LIN {X 0,Y 370.403,Z 508.31,A -85,B 0,C 180,E1 -12846.518,E2 -12846.518} C_VEL
LIN {X 0,Y 369.46,Z 515.734,A -85,B 0,C 180,E1 -12848.226,E2 -12848.226} C_VEL
LIN {X 0,Y 368.707,Z 521.584,A -85,B 0,C 180,E1 -12849.933,E2 -12849.933} C_VEL
LIN {X 0,Y 368.18,Z 526.14,A -85,B 0,C 180,E1 -12851.641,E2 -12851.641} C_VEL
LIN {X 0,Y 367.773,Z 529.554,A -85,B 0,C 180,E1 -12853.342,E2 -12853.342} C_VEL
LIN {X 0,Y 367.548,Z 531.232,A -85,B 0,C 180,E1 -12854.472,E2 -12854.472} C_VEL
LIN {X 0,Y 367.413,Z 532.492,A -85,B 0,C 180,E1 -12855.601,E2 -12855.601} C_VEL
LIN {X 0,Y 367.378,Z 533.578,A -85,B 0,C 180,E1 -12857.329,E2 -12857.329} C_VEL
LIN {X 0,Y 367.326,Z 533.705,A -85,B 0,C 180,E1 -12858.969,E2 -12858.969} C_VEL
LIN {X 0,Y 367.25,Z 533.313,A -85,B 0,C 180,E1 -12860.082,E2 -12860.082} C_VEL
LIN {X 0,Y 367.304,Z 532.493,A -85,B 0,C 180,E1 -12861.194,E2 -12861.194} C_VEL
LIN {X 0,Y 367.39,Z 531.247,A -85,B 0,C 180,E1 -12862.304,E2 -12862.304} C_VEL
LIN {X 0,Y 367.565,Z 528.8,A -85,B 0,C 180,E1 -12863.864,E2 -12863.864} C_VEL
LIN {X 0,Y 367.773,Z 524.966,A -85,B 0,C 180,E1 -12865.615,E2 -12865.615} C_VEL
LIN {X 0,Y 368.12,Z 520.21,A -85,B 0,C 180,E1 -12867.264,E2 -12867.264} C_VEL
LIN {X 0,Y 368.489,Z 514.221,A -85,B 0,C 180,E1 -12868.906,E2 -12868.906} C_VEL
LIN {X 0,Y 369.298,Z 506.742,A -85,B 0,C 180,E1 -12870.544,E2 -12870.544} C_VEL
LIN {X 0,Y 369.887,Z 499.149,A -85,B 0,C 180,E1 -12871.905,E2 -12871.905} C_VEL
LIN {X 0,Y 370.631,Z 489.936,A -85,B 0,C 180,E1 -12873.26,E2 -12873.26} C_VEL
LIN {X 0,Y 371.696,Z 479.626,A -85,B 0,C 180,E1 -12874.473,E2 -12874.473} C_VEL
LIN {X 0,Y 372.523,Z 468.25,A -85,B 0,C 180,E1 -12875.548,E2 -12875.548} C_VEL
LIN {X 0,Y 373.196,Z 456.407,A -85,B 0,C 180,E1 -12876.419,E2 -12876.419} C_VEL
LIN {X 0,Y 373.788,Z 443.261,A -85,B 0,C 180,E1 -12877.121,E2 -12877.121} C_VEL
LIN {X 0,Y 374.267,Z 430.141,A -85,B 0,C 180,E1 -12877.586,E2 -12877.586} C_VEL
LIN {X 0,Y 375.188,Z 377.579,A -85,B 0,C 180,E1 -12878.607,E2 -12878.607} C_VEL
LIN {X 0,Y 374.513,Z 369.843,A -85,B 0,C 180,E1 -12878.79,E2 -12878.79} C_VEL
LIN {X 0,Y 372.713,Z 362.305,A -85,B 0,C 180,E1 -12879.023,E2 -12879.023} C_VEL
LIN {X 0,Y 368.624,Z 347.244,A -85,B 0,C 180,E1 -12879.519,E2 -12879.519} C_VEL
LIN {X 0,Y 364.25,Z 322.715,A -85,B 0,C 180,E1 -12880.254,E2 -12880.254} C_VEL
LIN {X 0,Y 362.06,Z 310.498,A -85,B 0,C 180,E1 -12883.469,E2 -12883.469} C_VEL
LIN {X 0,Y 361.922,Z 310.404,A -85,B 0,C 180,E1 -12887.914,E2 -12887.914} C_VEL
LIN {X 0,Y 361.861,Z 310.408,A -85,B 0,C 180,E1 -12891.654,E2 -12891.654} C_VEL
LIN {X 0,Y 361.866,Z 310.405,A -85,B 0,C 180,E1 -12895.294,E2 -12895.294} C_VEL
LIN {X 0,Y 361.855,Z 310.407,A -85,B 0,C 180,E1 -12899.072,E2 -12899.072} C_VEL
LIN {X 0,Y 361.845,Z 310.41,A -85,B 0,C 180,E1 -12902.944,E2 -12902.944} C_VEL
LIN {X 0,Y 361.861,Z 310.406,A -85,B 0,C 180,E1 -12905.636,E2 -12905.636} C_VEL
LIN {X 0,Y 361.822,Z 310.414,A -85,B 0,C 180,E1 -12909.017,E2 -12909.017} C_VEL
LIN {X 0,Y 361.825,Z 310.418,A -85,B 0,C 180,E1 -12912.829,E2 -12912.829} C_VEL
LIN {X 0,Y 361.809,Z 310.412,A -85,B 0,C 180,E1 -12915.946,E2 -12915.946} C_VEL
LIN {X 0,Y 361.805,Z 310.417,A -85,B 0,C 180,E1 -12919.248,E2 -12919.248} C_VEL
LIN {X 0,Y 361.855,Z 310.411,A -85,B 0,C 180,E1 -12922.98,E2 -12922.98} C_VEL
LIN {X 0,Y 361.851,Z 310.408,A -85,B 0,C 180,E1 -12926.63,E2 -12926.63} C_VEL
LIN {X 0,Y 361.84,Z 310.412,A -85,B 0,C 180,E1 -12929.668,E2 -12929.668} C_VEL
LIN {X 0,Y 361.846,Z 310.415,A -85,B 0,C 180,E1 -12933.466,E2 -12933.466} C_VEL
LIN {X 0,Y 361.866,Z 310.407,A -85,B 0,C 180,E1 -12937.143,E2 -12937.143} C_VEL
LIN {X 0,Y 361.851,Z 310.407,A -85,B 0,C 180,E1 -12940.72,E2 -12940.72} C_VEL
LIN {X 0,Y 361.87,Z 310.407,A -85,B 0,C 180,E1 -12944.222,E2 -12944.222} C_VEL
LIN {X 0,Y 361.955,Z 310.395,A -85,B 0,C 180,E1 -12946.526,E2 -12946.526} C_VEL
LIN {X 0,Y 361.985,Z 310.397,A -85,B 0,C 180,E1 -12949.936,E2 -12949.936} C_VEL
LIN {X 0,Y 362.112,Z 310.375,A -85,B 0,C 180,E1 -12953.312,E2 -12953.312} C_VEL
LIN {X 0,Y 362.259,Z 310.358,A -85,B 0,C 180,E1 -12957.776,E2 -12957.776} C_VEL
LIN {X 0,Y 362.256,Z 310.361,A -85,B 0,C 180,E1 -12962.224,E2 -12962.224} C_VEL
LIN {X 0,Y 362.132,Z 310.377,A -85,B 0,C 180,E1 -12966.687,E2 -12966.687} C_VEL
LIN {X 0,Y 361.99,Z 310.391,A -85,B 0,C 180,E1 -12970.063,E2 -12970.063} C_VEL
LIN {X 0,Y 361.99,Z 310.39,A -85,B 0,C 180,E1 -12973.899,E2 -12973.899} C_VEL
LIN {X 0,Y 361.92,Z 310.405,A -85,B 0,C 180,E1 -12976.934,E2 -12976.934} C_VEL
LIN {X 0,Y 361.878,Z 310.405,A -85,B 0,C 180,E1 -12980.461,E2 -12980.461} C_VEL
LIN {X 0,Y 361.885,Z 310.403,A -85,B 0,C 180,E1 -12984.113,E2 -12984.113} C_VEL
LIN {X 0,Y 361.894,Z 310.403,A -85,B 0,C 180,E1 -12987.78,E2 -12987.78} C_VEL
LIN {X 0,Y 361.84,Z 310.415,A -85,B 0,C 180,E1 -12991.286,E2 -12991.286} C_VEL
LIN {X 0,Y 361.847,Z 310.408,A -85,B 0,C 180,E1 -12994.281,E2 -12994.281} C_VEL
LIN {X 0,Y 361.854,Z 310.41,A -85,B 0,C 180,E1 -12997.223,E2 -12997.223} C_VEL
LIN {X 0,Y 361.824,Z 310.411,A -85,B 0,C 180,E1 -13000.755,E2 -13000.755} C_VEL
LIN {X 0,Y 361.811,Z 310.413,A -85,B 0,C 180,E1 -13004.369,E2 -13004.369} C_VEL
LIN {X 0,Y 361.827,Z 310.414,A -85,B 0,C 180,E1 -13007.57,E2 -13007.57} C_VEL
LIN {X 0,Y 361.86,Z 310.406,A -85,B 0,C 180,E1 -13010.975,E2 -13010.975} C_VEL
LIN {X 0,Y 361.87,Z 310.406,A -85,B 0,C 180,E1 -13014.656,E2 -13014.656} C_VEL
LIN {X 0,Y 361.835,Z 310.414,A -85,B 0,C 180,E1 -13018.372,E2 -13018.372} C_VEL
LIN {X 0,Y 361.952,Z 310.565,A -85,B 0,C 180,E1 -13021.358,E2 -13021.358} C_VEL
LIN {X 0,Y 364.453,Z 323.504,A -85,B 0,C 180,E1 -13024.593,E2 -13024.593} C_VEL
LIN {X 0,Y 365.003,Z 327.454,A -85,B 0,C 180,E1 -13025.546,E2 -13025.546} C_VEL
LIN {X 0,Y 363.879,Z 341.559,A -85,B 0,C 180,E1 -13028.752,E2 -13028.752} C_VEL
LIN {X 0,Y 368.641,Z 375.347,A -85,B 0,C 180,E1 -13029.684,E2 -13029.684} C_VEL
LIN {X 0,Y 367.485,Z 450.609,A -85,B 0,C 180,E1 -13031.173,E2 -13031.173} C_VEL
LIN {X 0,Y 366.806,Z 464.431,A -85,B 0,C 180,E1 -13031.68,E2 -13031.68} C_VEL
LIN {X 0,Y 366.164,Z 476.327,A -85,B 0,C 180,E1 -13032.333,E2 -13032.333} C_VEL
LIN {X 0,Y 365.186,Z 488.345,A -85,B 0,C 180,E1 -13033.222,E2 -13033.222} C_VEL
LIN {X 0,Y 364.18,Z 499.863,A -85,B 0,C 180,E1 -13034.326,E2 -13034.326} C_VEL
LIN {X 0,Y 363.351,Z 510.251,A -85,B 0,C 180,E1 -13035.581,E2 -13035.581} C_VEL
LIN {X 0,Y 362.546,Z 518.72,A -85,B 0,C 180,E1 -13036.835,E2 -13036.835} C_VEL
LIN {X 0,Y 361.668,Z 527.891,A -85,B 0,C 180,E1 -13038.512,E2 -13038.512} C_VEL
LIN {X 0,Y 361.119,Z 535.278,A -85,B 0,C 180,E1 -13040.196,E2 -13040.196} C_VEL
LIN {X 0,Y 360.776,Z 540.273,A -85,B 0,C 180,E1 -13041.6,E2 -13041.6} C_VEL
LIN {X 0,Y 360.497,Z 545.112,A -85,B 0,C 180,E1 -13043.284,E2 -13043.284} C_VEL
LIN {X 0,Y 360.367,Z 548.816,A -85,B 0,C 180,E1 -13044.966,E2 -13044.966} C_VEL
LIN {X 0,Y 360.302,Z 551.49,A -85,B 0,C 180,E1 -13046.646,E2 -13046.646} C_VEL
LIN {X 0,Y 360.278,Z 552.747,A -85,B 0,C 180,E1 -13047.765,E2 -13047.765} C_VEL
LIN {X 0,Y 360.32,Z 553.602,A -85,B 0,C 180,E1 -13048.883,E2 -13048.883} C_VEL
LIN {X 0,Y 360.359,Z 554.017,A -85,B 0,C 180,E1 -13050.001,E2 -13050.001} C_VEL
LIN {X 0,Y 360.316,Z 554.039,A -85,B 0,C 180,E1 -13051.118,E2 -13051.118} C_VEL
LIN {X 0,Y 360.296,Z 552.931,A -85,B 0,C 180,E1 -13053.356,E2 -13053.356} C_VEL
LIN {X 0,Y 360.349,Z 551.747,A -85,B 0,C 180,E1 -13054.475,E2 -13054.475} C_VEL
LIN {X 0,Y 360.432,Z 549.428,A -85,B 0,C 180,E1 -13056.044,E2 -13056.044} C_VEL
LIN {X 0,Y 360.708,Z 545.699,A -85,B 0,C 180,E1 -13057.84,E2 -13057.84} C_VEL
LIN {X 0,Y 361.206,Z 541.093,A -85,B 0,C 180,E1 -13059.52,E2 -13059.52} C_VEL
LIN {X 0,Y 361.996,Z 534.151,A -85,B 0,C 180,E1 -13061.479,E2 -13061.479} C_VEL
LIN {X 0,Y 363.051,Z 526.659,A -85,B 0,C 180,E1 -13063.148,E2 -13063.148} C_VEL
LIN {X 0,Y 364.276,Z 517.674,A -85,B 0,C 180,E1 -13064.754,E2 -13064.754} C_VEL
LIN {X 0,Y 365.395,Z 507.667,A -85,B 0,C 180,E1 -13066.195,E2 -13066.195} C_VEL
LIN {X 0,Y 366.771,Z 496.964,A -85,B 0,C 180,E1 -13067.422,E2 -13067.422} C_VEL
LIN {X 0,Y 367.916,Z 486.591,A -85,B 0,C 180,E1 -13068.373,E2 -13068.373} C_VEL
LIN {X 0,Y 369.082,Z 474.147,A -85,B 0,C 180,E1 -13069.249,E2 -13069.249} C_VEL
LIN {X 0,Y 370.137,Z 461.039,A -85,B 0,C 180,E1 -13069.913,E2 -13069.913} C_VEL
LIN {X 0,Y 370.753,Z 447.912,A -85,B 0,C 180,E1 -13070.349,E2 -13070.349} C_VEL
LIN {X 0,Y 372.058,Z 374.718,A -85,B 0,C 180,E1 -13071.804,E2 -13071.804} C_VEL
LIN {X 0,Y 368.369,Z 353.96,A -85,B 0,C 180,E1 -13072.514,E2 -13072.514} C_VEL
LIN {X 0,Y 365.665,Z 341.104,A -85,B 0,C 180,E1 -13073.018,E2 -13073.018} C_VEL
LIN {X 0,Y 366.495,Z 332.811,A -85,B 0,C 180,E1 -13074.954,E2 -13074.954} C_VEL
LIN {X 0,Y 365.054,Z 324.101,A -85,B 0,C 180,E1 -13077.209,E2 -13077.209} C_VEL
LIN {X 0,Y 362.976,Z 314.837,A -85,B 0,C 180,E1 -13079.739,E2 -13079.739} C_VEL
LIN {X 0,Y 361.886,Z 310.417,A -85,B 0,C 180,E1 -13081,E2 -13081} C_VEL
LIN {X 0,Y 361.856,Z 310.415,A -85,B 0,C 180,E1 -13084.281,E2 -13084.281} C_VEL
LIN {X 0,Y 361.863,Z 310.411,A -85,B 0,C 180,E1 -13087.223,E2 -13087.223} C_VEL
LIN {X 0,Y 361.833,Z 310.413,A -85,B 0,C 180,E1 -13090.755,E2 -13090.755} C_VEL
LIN {X 0,Y 361.818,Z 310.416,A -85,B 0,C 180,E1 -13094.369,E2 -13094.369} C_VEL
LIN {X 0,Y 361.836,Z 310.412,A -85,B 0,C 180,E1 -13097.569,E2 -13097.569} C_VEL
LIN {X 0,Y 361.831,Z 310.41,A -85,B 0,C 180,E1 -13100.982,E2 -13100.982} C_VEL
LIN {X 0,Y 361.876,Z 310.405,A -85,B 0,C 180,E1 -13104.656,E2 -13104.656} C_VEL
LIN {X 0,Y 361.839,Z 310.406,A -85,B 0,C 180,E1 -13108.371,E2 -13108.371} C_VEL
LIN {X 0,Y 361.867,Z 310.407,A -85,B 0,C 180,E1 -13110.952,E2 -13110.952} C_VEL
LIN {X 0,Y 361.903,Z 310.403,A -85,B 0,C 180,E1 -13114.708,E2 -13114.708} C_VEL
LIN {X 0,Y 361.862,Z 310.405,A -85,B 0,C 180,E1 -13118.345,E2 -13118.345} C_VEL
LIN {X 0,Y 361.922,Z 310.397,A -85,B 0,C 180,E1 -13122.085,E2 -13122.085} C_VEL
LIN {X 0,Y 361.963,Z 310.397,A -85,B 0,C 180,E1 -13125.38,E2 -13125.38} C_VEL
LIN {X 0,Y 361.972,Z 310.389,A -85,B 0,C 180,E1 -13128.805,E2 -13128.805} C_VEL
LIN {X 0,Y 362.096,Z 310.373,A -85,B 0,C 180,E1 -13132.192,E2 -13132.192} C_VEL
LIN {X 0,Y 362.11,Z 310.373,A -85,B 0,C 180,E1 -13134.431,E2 -13134.431} C_VEL
LIN {X 0,Y 362.272,Z 310.354,A -85,B 0,C 180,E1 -13137.777,E2 -13137.777} C_VEL
LIN {X 0,Y 362.383,Z 310.337,A -85,B 0,C 180,E1 -13140,E2 -13140} C_VEL
LIN {X 0,Y 362.274,Z 310.357,A -85,B 0,C 180,E1 -13142.224,E2 -13142.224} C_VEL
LIN {X 0,Y 362.137,Z 310.375,A -85,B 0,C 180,E1 -13146.687,E2 -13146.687} C_VEL
LIN {X 0,Y 362.002,Z 310.386,A -85,B 0,C 180,E1 -13150.063,E2 -13150.063} C_VEL
LIN {X 0,Y 362,Z 310.384,A -85,B 0,C 180,E1 -13153.899,E2 -13153.899} C_VEL
LIN {X 0,Y 361.931,Z 310.396,A -85,B 0,C 180,E1 -13156.934,E2 -13156.934} C_VEL
LIN {X 0,Y 361.889,Z 310.406,A -85,B 0,C 180,E1 -13160.461,E2 -13160.461} C_VEL
LIN {X 0,Y 361.896,Z 310.401,A -85,B 0,C 180,E1 -13164.113,E2 -13164.113} C_VEL
LIN {X 0,Y 361.867,Z 310.403,A -85,B 0,C 180,E1 -13167.783,E2 -13167.783} C_VEL
LIN {X 0,Y 361.85,Z 310.408,A -85,B 0,C 180,E1 -13171.285,E2 -13171.285} C_VEL
LIN {X 0,Y 361.857,Z 310.405,A -85,B 0,C 180,E1 -13174.281,E2 -13174.281} C_VEL
LIN {X 0,Y 361.865,Z 310.408,A -85,B 0,C 180,E1 -13177.223,E2 -13177.223} C_VEL
LIN {X 0,Y 361.834,Z 310.412,A -85,B 0,C 180,E1 -13180.754,E2 -13180.754} C_VEL
LIN {X 0,Y 361.82,Z 310.416,A -85,B 0,C 180,E1 -13184.369,E2 -13184.369} C_VEL
LIN {X 0,Y 361.833,Z 310.415,A -85,B 0,C 180,E1 -13187.569,E2 -13187.569} C_VEL
LIN {X 0,Y 361.847,Z 310.414,A -85,B 0,C 180,E1 -13191.572,E2 -13191.572} C_VEL
LIN {X 0,Y 361.872,Z 310.526,A -85,B 0,C 180,E1 -13192.43,E2 -13192.43} C_VEL
LIN {X 0,Y 364.541,Z 322.027,A -85,B 0,C 180,E1 -13195.706,E2 -13195.706} C_VEL
LIN {X 0,Y 364.836,Z 323.293,A -85,B 0,C 180,E1 -13195.984,E2 -13195.984} C_VEL
LIN {X 0,Y 368.886,Z 333.647,A -85,B 0,C 180,E1 -13196.521,E2 -13196.521} C_VEL
LIN {X 0,Y 372.595,Z 349.964,A -85,B 0,C 180,E1 -13197.144,E2 -13197.144} C_VEL
LIN {X 0,Y 370.932,Z 431.121,A -85,B 0,C 180,E1 -13198.762,E2 -13198.762} C_VEL
LIN {X 0,Y 370.343,Z 443.628,A -85,B 0,C 180,E1 -13199.217,E2 -13199.217} C_VEL
LIN {X 0,Y 369.431,Z 456.148,A -85,B 0,C 180,E1 -13199.883,E2 -13199.883} C_VEL
LIN {X 0,Y 368.5,Z 467.865,A -85,B 0,C 180,E1 -13200.743,E2 -13200.743} C_VEL
LIN {X 0,Y 367.446,Z 478.453,A -85,B 0,C 180,E1 -13201.741,E2 -13201.741} C_VEL
LIN {X 0,Y 366.088,Z 489.395,A -85,B 0,C 180,E1 -13203.028,E2 -13203.028} C_VEL
LIN {X 0,Y 364.922,Z 498.248,A -85,B 0,C 180,E1 -13204.321,E2 -13204.321} C_VEL
LIN {X 0,Y 363.845,Z 506.491,A -85,B 0,C 180,E1 -13205.796,E2 -13205.796} C_VEL
LIN {X 0,Y 362.75,Z 514.16,A -85,B 0,C 180,E1 -13207.502,E2 -13207.502} C_VEL
LIN {X 0,Y 361.981,Z 519.921,A -85,B 0,C 180,E1 -13209.097,E2 -13209.097} C_VEL
LIN {X 0,Y 361.351,Z 524.542,A -85,B 0,C 180,E1 -13210.692,E2 -13210.692} C_VEL
LIN {X 0,Y 360.86,Z 528.773,A -85,B 0,C 180,E1 -13212.615,E2 -13212.615} C_VEL
LIN {X 0,Y 360.531,Z 531.23,A -85,B 0,C 180,E1 -13214.162,E2 -13214.162} C_VEL
LIN {X 0,Y 360.351,Z 532.536,A -85,B 0,C 180,E1 -13215.312,E2 -13215.312} C_VEL
LIN {X 0,Y 360.305,Z 533.779,A -85,B 0,C 180,E1 -13217.238,E2 -13217.238} C_VEL
LIN {X 0,Y 360.227,Z 533.928,A -85,B 0,C 180,E1 -13218.749,E2 -13218.749} C_VEL
LIN {X 0,Y 360.191,Z 532.839,A -85,B 0,C 180,E1 -13221.019,E2 -13221.019} C_VEL
LIN {X 0,Y 360.283,Z 531.649,A -85,B 0,C 180,E1 -13222.151,E2 -13222.151} C_VEL
LIN {X 0,Y 360.472,Z 528.995,A -85,B 0,C 180,E1 -13223.901,E2 -13223.901} C_VEL
LIN {X 0,Y 360.69,Z 525.557,A -85,B 0,C 180,E1 -13225.529,E2 -13225.529} C_VEL
LIN {X 0,Y 361.026,Z 520.906,A -85,B 0,C 180,E1 -13227.21,E2 -13227.21} C_VEL
LIN {X 0,Y 361.5,Z 513.916,A -85,B 0,C 180,E1 -13229.164,E2 -13229.164} C_VEL
LIN {X 0,Y 362.336,Z 506.326,A -85,B 0,C 180,E1 -13230.833,E2 -13230.833} C_VEL
LIN {X 0,Y 362.951,Z 498.598,A -85,B 0,C 180,E1 -13232.219,E2 -13232.219} C_VEL
LIN {X 0,Y 363.778,Z 489.158,A -85,B 0,C 180,E1 -13233.599,E2 -13233.599} C_VEL
LIN {X 0,Y 364.871,Z 478.645,A -85,B 0,C 180,E1 -13234.833,E2 -13234.833} C_VEL
LIN {X 0,Y 365.739,Z 466.986,A -85,B 0,C 180,E1 -13235.928,E2 -13235.928} C_VEL
LIN {X 0,Y 366.426,Z 454.561,A -85,B 0,C 180,E1 -13236.815,E2 -13236.815} C_VEL
LIN {X 0,Y 367.031,Z 441.442,A -85,B 0,C 180,E1 -13237.495,E2 -13237.495} C_VEL
LIN {X 0,Y 367.466,Z 429.535,A -85,B 0,C 180,E1 -13237.9,E2 -13237.9} C_VEL
LIN {X 0,Y 368.821,Z 348.26,A -85,B 0,C 180,E1 -13239.489,E2 -13239.489} C_VEL
LIN {X 0,Y 368.624,Z 347.244,A -85,B 0,C 180,E1 -13239.519,E2 -13239.519} C_VEL
LIN {X 0,Y 367.316,Z 343.592,A -85,B 0,C 180,E1 -13239.657,E2 -13239.657} C_VEL
LIN {X 0,Y 360.025,Z 332.897,A -85,B 0,C 180,E1 -13240.245,E2 -13240.245} C_VEL
LIN {X 0,Y 358.636,Z 329.265,A -85,B 0,C 180,E1 -13240.392,E2 -13240.392} C_VEL
LIN {X 0,Y 357.145,Z 322.897,A -85,B 0,C 180,E1 -13240.626,E2 -13240.626} C_VEL
LIN {X 0,Y 354.977,Z 311.27,A -85,B 0,C 180,E1 -13243.783,E2 -13243.783} C_VEL
LIN {X 0,Y 354.891,Z 311.28,A -85,B 0,C 180,E1 -13248.091,E2 -13248.091} C_VEL
LIN {X 0,Y 354.815,Z 311.29,A -85,B 0,C 180,E1 -13252.106,E2 -13252.106} C_VEL
LIN {X 0,Y 354.802,Z 311.287,A -85,B 0,C 180,E1 -13255.834,E2 -13255.834} C_VEL
LIN {X 0,Y 354.792,Z 311.287,A -85,B 0,C 180,E1 -13259.683,E2 -13259.683} C_VEL
LIN {X 0,Y 354.783,Z 311.293,A -85,B 0,C 180,E1 -13262.332,E2 -13262.332} C_VEL
LIN {X 0,Y 354.816,Z 311.284,A -85,B 0,C 180,E1 -13265.697,E2 -13265.697} C_VEL
LIN {X 0,Y 354.765,Z 311.29,A -85,B 0,C 180,E1 -13269.411,E2 -13269.411} C_VEL
LIN {X 0,Y 354.777,Z 311.295,A -85,B 0,C 180,E1 -13272.865,E2 -13272.865} C_VEL
LIN {X 0,Y 354.758,Z 311.291,A -85,B 0,C 180,E1 -13276.102,E2 -13276.102} C_VEL
LIN {X 0,Y 354.758,Z 311.296,A -85,B 0,C 180,E1 -13279.174,E2 -13279.174} C_VEL
LIN {X 0,Y 354.793,Z 311.287,A -85,B 0,C 180,E1 -13282.403,E2 -13282.403} C_VEL
LIN {X 0,Y 354.802,Z 311.289,A -85,B 0,C 180,E1 -13284.939,E2 -13284.939} C_VEL
LIN {X 0,Y 354.769,Z 311.289,A -85,B 0,C 180,E1 -13288.409,E2 -13288.409} C_VEL
LIN {X 0,Y 354.781,Z 311.293,A -85,B 0,C 180,E1 -13291.613,E2 -13291.613} C_VEL
LIN {X 0,Y 354.798,Z 311.291,A -85,B 0,C 180,E1 -13295.419,E2 -13295.419} C_VEL
LIN {X 0,Y 354.816,Z 311.285,A -85,B 0,C 180,E1 -13299.112,E2 -13299.112} C_VEL
LIN {X 0,Y 354.836,Z 311.281,A -85,B 0,C 180,E1 -13302.716,E2 -13302.716} C_VEL
LIN {X 0,Y 354.9,Z 311.276,A -85,B 0,C 180,E1 -13306.253,E2 -13306.253} C_VEL
LIN {X 0,Y 354.941,Z 311.272,A -85,B 0,C 180,E1 -13309.735,E2 -13309.735} C_VEL
LIN {X 0,Y 355.078,Z 311.251,A -85,B 0,C 180,E1 -13313.179,E2 -13313.179} C_VEL
LIN {X 0,Y 355.221,Z 311.235,A -85,B 0,C 180,E1 -13317.732,E2 -13317.732} C_VEL
LIN {X 0,Y 355.162,Z 311.241,A -85,B 0,C 180,E1 -13321.134,E2 -13321.134} C_VEL
LIN {X 0,Y 355.219,Z 311.239,A -85,B 0,C 180,E1 -13322.268,E2 -13322.268} C_VEL
LIN {X 0,Y 355.096,Z 311.252,A -85,B 0,C 180,E1 -13326.82,E2 -13326.82} C_VEL
LIN {X 0,Y 354.946,Z 311.27,A -85,B 0,C 180,E1 -13330.265,E2 -13330.265} C_VEL
LIN {X 0,Y 354.934,Z 311.269,A -85,B 0,C 180,E1 -13334.019,E2 -13334.019} C_VEL
LIN {X 0,Y 354.882,Z 311.275,A -85,B 0,C 180,E1 -13338.092,E2 -13338.092} C_VEL
LIN {X 0,Y 354.807,Z 311.285,A -85,B 0,C 180,E1 -13342.108,E2 -13342.108} C_VEL
LIN {X 0,Y 354.868,Z 311.278,A -85,B 0,C 180,E1 -13345.83,E2 -13345.83} C_VEL
LIN {X 0,Y 354.811,Z 311.287,A -85,B 0,C 180,E1 -13349.682,E2 -13349.682} C_VEL
LIN {X 0,Y 354.799,Z 311.289,A -85,B 0,C 180,E1 -13353.703,E2 -13353.703} C_VEL
LIN {X 0,Y 354.789,Z 311.287,A -85,B 0,C 180,E1 -13356.46,E2 -13356.46} C_VEL
LIN {X 0,Y 354.792,Z 311.291,A -85,B 0,C 180,E1 -13359.419,E2 -13359.419} C_VEL
LIN {X 0,Y 354.78,Z 311.288,A -85,B 0,C 180,E1 -13362.868,E2 -13362.868} C_VEL
LIN {X 0,Y 354.762,Z 311.294,A -85,B 0,C 180,E1 -13366.105,E2 -13366.105} C_VEL
LIN {X 0,Y 354.777,Z 311.289,A -85,B 0,C 180,E1 -13369.179,E2 -13369.179} C_VEL
LIN {X 0,Y 354.802,Z 311.288,A -85,B 0,C 180,E1 -13372.404,E2 -13372.404} C_VEL
LIN {X 0,Y 354.808,Z 311.285,A -85,B 0,C 180,E1 -13374.942,E2 -13374.942} C_VEL
LIN {X 0,Y 354.79,Z 311.291,A -85,B 0,C 180,E1 -13378.406,E2 -13378.406} C_VEL
LIN {X 0,Y 354.903,Z 311.437,A -85,B 0,C 180,E1 -13381.089,E2 -13381.089} C_VEL
LIN {X 0,Y 357.176,Z 322.947,A -85,B 0,C 180,E1 -13384.037,E2 -13384.037} C_VEL
LIN {X 0,Y 358.032,Z 328.399,A -85,B 0,C 180,E1 -13385.389,E2 -13385.389} C_VEL
LIN {X 0,Y 356.944,Z 341.426,A -85,B 0,C 180,E1 -13388.407,E2 -13388.407} C_VEL
LIN {X 0,Y 361.841,Z 375.651,A -85,B 0,C 180,E1 -13389.364,E2 -13389.364} C_VEL
LIN {X 0,Y 360.697,Z 449.455,A -85,B 0,C 180,E1 -13390.842,E2 -13390.842} C_VEL
LIN {X 0,Y 360.099,Z 462.843,A -85,B 0,C 180,E1 -13391.326,E2 -13391.326} C_VEL
LIN {X 0,Y 359.327,Z 475.085,A -85,B 0,C 180,E1 -13391.986,E2 -13391.986} C_VEL
LIN {X 0,Y 358.384,Z 487.421,A -85,B 0,C 180,E1 -13392.894,E2 -13392.894} C_VEL
LIN {X 0,Y 357.287,Z 499.066,A -85,B 0,C 180,E1 -13394.016,E2 -13394.016} C_VEL
LIN {X 0,Y 356.437,Z 509.566,A -85,B 0,C 180,E1 -13395.295,E2 -13395.295} C_VEL
LIN {X 0,Y 355.561,Z 518.122,A -85,B 0,C 180,E1 -13396.571,E2 -13396.571} C_VEL
LIN {X 0,Y 354.837,Z 526.007,A -85,B 0,C 180,E1 -13397.998,E2 -13397.998} C_VEL
LIN {X 0,Y 354.166,Z 533.693,A -85,B 0,C 180,E1 -13399.713,E2 -13399.713} C_VEL
LIN {X 0,Y 353.709,Z 539.865,A -85,B 0,C 180,E1 -13401.431,E2 -13401.431} C_VEL
LIN {X 0,Y 353.415,Z 544.75,A -85,B 0,C 180,E1 -13403.148,E2 -13403.148} C_VEL
LIN {X 0,Y 353.269,Z 548.496,A -85,B 0,C 180,E1 -13404.865,E2 -13404.865} C_VEL
LIN {X 0,Y 353.224,Z 551.21,A -85,B 0,C 180,E1 -13406.579,E2 -13406.579} C_VEL
LIN {X 0,Y 353.221,Z 553.365,A -85,B 0,C 180,E1 -13408.861,E2 -13408.861} C_VEL
LIN {X 0,Y 353.262,Z 553.809,A -85,B 0,C 180,E1 -13410.001,E2 -13410.001} C_VEL
LIN {X 0,Y 353.215,Z 553.849,A -85,B 0,C 180,E1 -13411.141,E2 -13411.141} C_VEL
LIN {X 0,Y 353.218,Z 552.78,A -85,B 0,C 180,E1 -13413.423,E2 -13413.423} C_VEL
LIN {X 0,Y 353.263,Z 551.63,A -85,B 0,C 180,E1 -13414.565,E2 -13414.565} C_VEL
LIN {X 0,Y 353.324,Z 549.627,A -85,B 0,C 180,E1 -13415.98,E2 -13415.98} C_VEL
LIN {X 0,Y 353.675,Z 545.653,A -85,B 0,C 180,E1 -13417.996,E2 -13417.996} C_VEL
LIN {X 0,Y 354.165,Z 541.091,A -85,B 0,C 180,E1 -13419.711,E2 -13419.711} C_VEL
LIN {X 0,Y 354.998,Z 534.204,A -85,B 0,C 180,E1 -13421.709,E2 -13421.709} C_VEL
LIN {X 0,Y 356.126,Z 526.766,A -85,B 0,C 180,E1 -13423.409,E2 -13423.409} C_VEL
LIN {X 0,Y 357.402,Z 518.024,A -85,B 0,C 180,E1 -13425.019,E2 -13425.019} C_VEL
LIN {X 0,Y 358.456,Z 509.016,A -85,B 0,C 180,E1 -13426.371,E2 -13426.371} C_VEL
LIN {X 0,Y 359.852,Z 498.64,A -85,B 0,C 180,E1 -13427.622,E2 -13427.622} C_VEL
LIN {X 0,Y 361.227,Z 487.135,A -85,B 0,C 180,E1 -13428.725,E2 -13428.725} C_VEL
LIN {X 0,Y 362.434,Z 475,A -85,B 0,C 180,E1 -13429.616,E2 -13429.616} C_VEL
LIN {X 0,Y 363.538,Z 462.262,A -85,B 0,C 180,E1 -13430.291,E2 -13430.291} C_VEL
LIN {X 0,Y 364.234,Z 448.972,A -85,B 0,C 180,E1 -13430.767,E2 -13430.767} C_VEL
LIN {X 0,Y 365.682,Z 375.911,A -85,B 0,C 180,E1 -13432.246,E2 -13432.246} C_VEL
LIN {X 0,Y 362.041,Z 355.49,A -85,B 0,C 180,E1 -13432.965,E2 -13432.965} C_VEL
LIN {X 0,Y 358.953,Z 340.869,A -85,B 0,C 180,E1 -13433.558,E2 -13433.558} C_VEL
LIN {X 0,Y 359.615,Z 334.178,A -85,B 0,C 180,E1 -13435.155,E2 -13435.155} C_VEL
LIN {X 0,Y 358.206,Z 325.788,A -85,B 0,C 180,E1 -13437.378,E2 -13437.378} C_VEL
LIN {X 0,Y 355.847,Z 315.566,A -85,B 0,C 180,E1 -13440.245,E2 -13440.245} C_VEL
LIN {X 0,Y 354.805,Z 311.295,A -85,B 0,C 180,E1 -13441.493,E2 -13441.493} C_VEL
LIN {X 0,Y 354.814,Z 311.292,A -85,B 0,C 180,E1 -13445.06,E2 -13445.06} C_VEL
LIN {X 0,Y 354.798,Z 311.29,A -85,B 0,C 180,E1 -13447.884,E2 -13447.884} C_VEL
LIN {X 0,Y 354.785,Z 311.289,A -85,B 0,C 180,E1 -13451.171,E2 -13451.171} C_VEL
LIN {X 0,Y 354.765,Z 311.296,A -85,B 0,C 180,E1 -13454.506,E2 -13454.506} C_VEL
LIN {X 0,Y 354.794,Z 311.289,A -85,B 0,C 180,E1 -13457.663,E2 -13457.663} C_VEL
LIN {X 0,Y 354.786,Z 311.291,A -85,B 0,C 180,E1 -13460.662,E2 -13460.662} C_VEL
LIN {X 0,Y 354.823,Z 311.284,A -85,B 0,C 180,E1 -13464.301,E2 -13464.301} C_VEL
LIN {X 0,Y 354.788,Z 311.284,A -85,B 0,C 180,E1 -13467.667,E2 -13467.667} C_VEL
LIN {X 0,Y 354.812,Z 311.283,A -85,B 0,C 180,E1 -13471.616,E2 -13471.616} C_VEL
LIN {X 0,Y 354.855,Z 311.279,A -85,B 0,C 180,E1 -13475.423,E2 -13475.423} C_VEL
LIN {X 0,Y 354.828,Z 311.281,A -85,B 0,C 180,E1 -13479.113,E2 -13479.113} C_VEL
LIN {X 0,Y 354.881,Z 311.274,A -85,B 0,C 180,E1 -13482.719,E2 -13482.719} C_VEL
LIN {X 0,Y 354.953,Z 311.264,A -85,B 0,C 180,E1 -13486.255,E2 -13486.255} C_VEL
LIN {X 0,Y 354.977,Z 311.266,A -85,B 0,C 180,E1 -13489.736,E2 -13489.736} C_VEL
LIN {X 0,Y 355.112,Z 311.243,A -85,B 0,C 180,E1 -13493.18,E2 -13493.18} C_VEL
LIN {X 0,Y 355.234,Z 311.23,A -85,B 0,C 180,E1 -13497.733,E2 -13497.733} C_VEL
LIN {X 0,Y 355.334,Z 311.215,A -85,B 0,C 180,E1 -13500,E2 -13500} C_VEL
LIN {X 0,Y 355.236,Z 311.234,A -85,B 0,C 180,E1 -13502.268,E2 -13502.268} C_VEL
LIN {X 0,Y 355.101,Z 311.25,A -85,B 0,C 180,E1 -13506.82,E2 -13506.82} C_VEL
LIN {X 0,Y 354.958,Z 311.265,A -85,B 0,C 180,E1 -13510.265,E2 -13510.265} C_VEL
LIN {X 0,Y 354.945,Z 311.263,A -85,B 0,C 180,E1 -13514.019,E2 -13514.019} C_VEL
LIN {X 0,Y 354.892,Z 311.269,A -85,B 0,C 180,E1 -13518.092,E2 -13518.092} C_VEL
LIN {X 0,Y 354.821,Z 311.279,A -85,B 0,C 180,E1 -13521.418,E2 -13521.418} C_VEL
LIN {X 0,Y 354.856,Z 311.279,A -85,B 0,C 180,E1 -13524.577,E2 -13524.577} C_VEL
LIN {X 0,Y 354.813,Z 311.281,A -85,B 0,C 180,E1 -13528.385,E2 -13528.385} C_VEL
LIN {X 0,Y 354.79,Z 311.286,A -85,B 0,C 180,E1 -13532.334,E2 -13532.334} C_VEL
LIN {X 0,Y 354.825,Z 311.288,A -85,B 0,C 180,E1 -13535.699,E2 -13535.699} C_VEL
LIN {X 0,Y 354.828,Z 311.286,A -85,B 0,C 180,E1 -13539.424,E2 -13539.424} C_VEL
LIN {X 0,Y 354.79,Z 311.29,A -85,B 0,C 180,E1 -13542.867,E2 -13542.867} C_VEL
LIN {X 0,Y 354.769,Z 311.294,A -85,B 0,C 180,E1 -13546.103,E2 -13546.103} C_VEL
LIN {X 0,Y 354.769,Z 311.292,A -85,B 0,C 180,E1 -13549.176,E2 -13549.176} C_VEL
LIN {X 0,Y 354.838,Z 311.372,A -85,B 0,C 180,E1 -13551.941,E2 -13551.941} C_VEL
LIN {X 0,Y 357.414,Z 322.648,A -85,B 0,C 180,E1 -13555.232,E2 -13555.232} C_VEL
LIN {X 0,Y 357.63,Z 323.461,A -85,B 0,C 180,E1 -13555.404,E2 -13555.404} C_VEL
LIN {X 0,Y 362.707,Z 335.781,A -85,B 0,C 180,E1 -13556.087,E2 -13556.087} C_VEL
LIN {X 0,Y 366.192,Z 350.851,A -85,B 0,C 180,E1 -13556.683,E2 -13556.683} C_VEL
LIN {X 0,Y 364.501,Z 430.652,A -85,B 0,C 180,E1 -13558.295,E2 -13558.295} C_VEL
LIN {X 0,Y 363.883,Z 442.839,A -85,B 0,C 180,E1 -13558.73,E2 -13558.73} C_VEL
LIN {X 0,Y 362.895,Z 456.195,A -85,B 0,C 180,E1 -13559.444,E2 -13559.444} C_VEL
LIN {X 0,Y 361.93,Z 467.953,A -85,B 0,C 180,E1 -13560.319,E2 -13560.319} C_VEL
LIN {X 0,Y 360.782,Z 478.764,A -85,B 0,C 180,E1 -13561.355,E2 -13561.355} C_VEL
LIN {X 0,Y 359.372,Z 489.502,A -85,B 0,C 180,E1 -13562.64,E2 -13562.64} C_VEL
LIN {X 0,Y 358.032,Z 499.267,A -85,B 0,C 180,E1 -13564.102,E2 -13564.102} C_VEL
LIN {X 0,Y 356.934,Z 507.189,A -85,B 0,C 180,E1 -13565.575,E2 -13565.575} C_VEL
LIN {X 0,Y 355.785,Z 514.882,A -85,B 0,C 180,E1 -13567.344,E2 -13567.344} C_VEL
LIN {X 0,Y 354.918,Z 521.01,A -85,B 0,C 180,E1 -13569.118,E2 -13569.118} C_VEL
LIN {X 0,Y 354.218,Z 525.801,A -85,B 0,C 180,E1 -13570.89,E2 -13570.89} C_VEL
LIN {X 0,Y 353.77,Z 529.418,A -85,B 0,C 180,E1 -13572.662,E2 -13572.662} C_VEL
LIN {X 0,Y 353.504,Z 531.23,A -85,B 0,C 180,E1 -13573.839,E2 -13573.839} C_VEL
LIN {X 0,Y 353.3,Z 532.581,A -85,B 0,C 180,E1 -13575.012,E2 -13575.012} C_VEL
LIN {X 0,Y 353.204,Z 533.989,A -85,B 0,C 180,E1 -13577.162,E2 -13577.162} C_VEL
LIN {X 0,Y 353.133,Z 534.151,A -85,B 0,C 180,E1 -13578.52,E2 -13578.52} C_VEL
LIN {X 0,Y 353.096,Z 533.15,A -85,B 0,C 180,E1 -13580.837,E2 -13580.837} C_VEL
LIN {X 0,Y 353.171,Z 532.046,A -85,B 0,C 180,E1 -13581.992,E2 -13581.992} C_VEL
LIN {X 0,Y 353.379,Z 529.183,A -85,B 0,C 180,E1 -13583.939,E2 -13583.939} C_VEL
LIN {X 0,Y 353.605,Z 526.126,A -85,B 0,C 180,E1 -13585.439,E2 -13585.439} C_VEL
LIN {X 0,Y 353.931,Z 521.585,A -85,B 0,C 180,E1 -13587.154,E2 -13587.154} C_VEL
LIN {X 0,Y 354.389,Z 514.719,A -85,B 0,C 180,E1 -13589.147,E2 -13589.147} C_VEL
LIN {X 0,Y 355.259,Z 507.258,A -85,B 0,C 180,E1 -13590.849,E2 -13590.849} C_VEL
LIN {X 0,Y 355.888,Z 499.686,A -85,B 0,C 180,E1 -13592.263,E2 -13592.263} C_VEL
LIN {X 0,Y 356.692,Z 490.51,A -85,B 0,C 180,E1 -13593.671,E2 -13593.671} C_VEL
LIN {X 0,Y 357.839,Z 480.233,A -85,B 0,C 180,E1 -13594.928,E2 -13594.928} C_VEL
LIN {X 0,Y 358.723,Z 468.904,A -85,B 0,C 180,E1 -13596.044,E2 -13596.044} C_VEL
LIN {X 0,Y 359.444,Z 457.152,A -85,B 0,C 180,E1 -13596.948,E2 -13596.948} C_VEL
LIN {X 0,Y 360.083,Z 444.157,A -85,B 0,C 180,E1 -13597.675,E2 -13597.675} C_VEL
LIN {X 0,Y 360.582,Z 431.295,A -85,B 0,C 180,E1 -13598.158,E2 -13598.158} C_VEL
LIN {X 0,Y 361.332,Z 396.081,A -85,B 0,C 180,E1 -13598.88,E2 -13598.88} C_VEL
LIN {X 0,Y 362.108,Z 349.433,A -85,B 0,C 180,E1 -13599.798,E2 -13599.798} C_VEL
LIN {X 0,Y 358.636,Z 329.265,A -85,B 0,C 180,E1 -13600.392,E2 -13600.392} C_VEL
LIN {X 0,Y 357.479,Z 326.375,A -85,B 0,C 180,E1 -13600.564,E2 -13600.564} C_VEL
LIN {X 0,Y 354.976,Z 323.264,A -85,B 0,C 180,E1 -13600.966,E2 -13600.966} C_VEL
LIN {X 0,Y 351.853,Z 320.629,A -85,B 0,C 180,E1 -13601.58,E2 -13601.58} C_VEL
LIN {X 0,Y 349.414,Z 318.229,A -85,B 0,C 180,E1 -13602.314,E2 -13602.314} C_VEL
LIN {X 0,Y 348.844,Z 316.873,A -85,B 0,C 180,E1 -13602.707,E2 -13602.707} C_VEL
LIN {X 0,Y 347.895,Z 312.152,A -85,B 0,C 180,E1 -13604.028,E2 -13604.028} C_VEL
LIN {X 0,Y 347.83,Z 312.158,A -85,B 0,C 180,E1 -13608.258,E2 -13608.258} C_VEL
LIN {X 0,Y 347.768,Z 312.163,A -85,B 0,C 180,E1 -13611.625,E2 -13611.625} C_VEL
LIN {X 0,Y 347.739,Z 312.165,A -85,B 0,C 180,E1 -13615.113,E2 -13615.113} C_VEL
LIN {X 0,Y 347.728,Z 312.167,A -85,B 0,C 180,E1 -13617.7,E2 -13617.7} C_VEL
LIN {X 0,Y 347.734,Z 312.172,A -85,B 0,C 180,E1 -13620.348,E2 -13620.348} C_VEL
LIN {X 0,Y 347.746,Z 312.166,A -85,B 0,C 180,E1 -13624.042,E2 -13624.042} C_VEL
LIN {X 0,Y 347.752,Z 312.164,A -85,B 0,C 180,E1 -13627.32,E2 -13627.32} C_VEL
LIN {X 0,Y 347.693,Z 312.173,A -85,B 0,C 180,E1 -13630.301,E2 -13630.301} C_VEL
LIN {X 0,Y 347.717,Z 312.169,A -85,B 0,C 180,E1 -13633.407,E2 -13633.407} C_VEL
LIN {X 0,Y 347.718,Z 312.171,A -85,B 0,C 180,E1 -13636.686,E2 -13636.686} C_VEL
LIN {X 0,Y 347.696,Z 312.171,A -85,B 0,C 180,E1 -13640.181,E2 -13640.181} C_VEL
LIN {X 0,Y 347.749,Z 312.166,A -85,B 0,C 180,E1 -13642.677,E2 -13642.677} C_VEL
LIN {X 0,Y 347.742,Z 312.165,A -85,B 0,C 180,E1 -13645.955,E2 -13645.955} C_VEL
LIN {X 0,Y 347.719,Z 312.171,A -85,B 0,C 180,E1 -13649.649,E2 -13649.649} C_VEL
LIN {X 0,Y 347.728,Z 312.172,A -85,B 0,C 180,E1 -13653.599,E2 -13653.599} C_VEL
LIN {X 0,Y 347.744,Z 312.166,A -85,B 0,C 180,E1 -13656.158,E2 -13656.158} C_VEL
LIN {X 0,Y 347.768,Z 312.166,A -85,B 0,C 180,E1 -13659.906,E2 -13659.906} C_VEL
LIN {X 0,Y 347.778,Z 312.164,A -85,B 0,C 180,E1 -13663.565,E2 -13663.565} C_VEL
LIN {X 0,Y 347.855,Z 312.151,A -85,B 0,C 180,E1 -13667.159,E2 -13667.159} C_VEL
LIN {X 0,Y 347.925,Z 312.143,A -85,B 0,C 180,E1 -13670.7,E2 -13670.7} C_VEL
LIN {X 0,Y 348.028,Z 312.135,A -85,B 0,C 180,E1 -13674.205,E2 -13674.205} C_VEL
LIN {X 0,Y 348.183,Z 312.111,A -85,B 0,C 180,E1 -13677.686,E2 -13677.686} C_VEL
LIN {X 0,Y 348.131,Z 312.117,A -85,B 0,C 180,E1 -13681.157,E2 -13681.157} C_VEL
LIN {X 0,Y 348.18,Z 312.116,A -85,B 0,C 180,E1 -13682.313,E2 -13682.313} C_VEL
LIN {X 0,Y 348.063,Z 312.127,A -85,B 0,C 180,E1 -13686.958,E2 -13686.958} C_VEL
LIN {X 0,Y 347.887,Z 312.151,A -85,B 0,C 180,E1 -13690.475,E2 -13690.475} C_VEL
LIN {X 0,Y 347.891,Z 312.147,A -85,B 0,C 180,E1 -13694.15,E2 -13694.15} C_VEL
LIN {X 0,Y 347.821,Z 312.156,A -85,B 0,C 180,E1 -13698.259,E2 -13698.259} C_VEL
LIN {X 0,Y 347.759,Z 312.164,A -85,B 0,C 180,E1 -13701.626,E2 -13701.626} C_VEL
LIN {X 0,Y 347.792,Z 312.165,A -85,B 0,C 180,E1 -13705.11,E2 -13705.11} C_VEL
LIN {X 0,Y 347.795,Z 312.16,A -85,B 0,C 180,E1 -13707.695,E2 -13707.695} C_VEL
LIN {X 0,Y 347.742,Z 312.165,A -85,B 0,C 180,E1 -13710.349,E2 -13710.349} C_VEL
LIN {X 0,Y 347.742,Z 312.166,A -85,B 0,C 180,E1 -13714.044,E2 -13714.044} C_VEL
LIN {X 0,Y 347.75,Z 312.168,A -85,B 0,C 180,E1 -13717.322,E2 -13717.322} C_VEL
LIN {X 0,Y 347.713,Z 312.169,A -85,B 0,C 180,E1 -13720.3,E2 -13720.3} C_VEL
LIN {X 0,Y 347.717,Z 312.171,A -85,B 0,C 180,E1 -13723.409,E2 -13723.409} C_VEL
LIN {X 0,Y 347.719,Z 312.168,A -85,B 0,C 180,E1 -13726.687,E2 -13726.687} C_VEL
LIN {X 0,Y 347.742,Z 312.169,A -85,B 0,C 180,E1 -13730.174,E2 -13730.174} C_VEL
LIN {X 0,Y 347.757,Z 312.164,A -85,B 0,C 180,E1 -13732.68,E2 -13732.68} C_VEL
LIN {X 0,Y 347.745,Z 312.169,A -85,B 0,C 180,E1 -13735.957,E2 -13735.957} C_VEL
LIN {X 0,Y 347.758,Z 312.164,A -85,B 0,C 180,E1 -13739.654,E2 -13739.654} C_VEL
LIN {X 0,Y 347.831,Z 312.263,A -85,B 0,C 180,E1 -13740.797,E2 -13740.797} C_VEL
LIN {X 0,Y 350.102,Z 323.703,A -85,B 0,C 180,E1 -13743.793,E2 -13743.793} C_VEL
LIN {X 0,Y 351.055,Z 330.297,A -85,B 0,C 180,E1 -13745.456,E2 -13745.456} C_VEL
LIN {X 0,Y 350.058,Z 341.235,A -85,B 0,C 180,E1 -13748.038,E2 -13748.038} C_VEL
LIN {X 0,Y 355.07,Z 376.183,A -85,B 0,C 180,E1 -13749.038,E2 -13749.038} C_VEL
LIN {X 0,Y 353.88,Z 449.425,A -85,B 0,C 180,E1 -13750.534,E2 -13750.534} C_VEL
LIN {X 0,Y 353.266,Z 462.76,A -85,B 0,C 180,E1 -13751.027,E2 -13751.027} C_VEL
LIN {X 0,Y 352.455,Z 474.974,A -85,B 0,C 180,E1 -13751.697,E2 -13751.697} C_VEL
LIN {X 0,Y 351.53,Z 486.474,A -85,B 0,C 180,E1 -13752.55,E2 -13752.55} C_VEL
LIN {X 0,Y 350.394,Z 498.267,A -85,B 0,C 180,E1 -13753.693,E2 -13753.693} C_VEL
LIN {X 0,Y 349.528,Z 508.944,A -85,B 0,C 180,E1 -13755.007,E2 -13755.007} C_VEL
LIN {X 0,Y 348.609,Z 517.512,A -85,B 0,C 180,E1 -13756.298,E2 -13756.298} C_VEL
LIN {X 0,Y 347.854,Z 525.476,A -85,B 0,C 180,E1 -13757.753,E2 -13757.753} C_VEL
LIN {X 0,Y 347.136,Z 533.236,A -85,B 0,C 180,E1 -13759.502,E2 -13759.502} C_VEL
LIN {X 0,Y 346.661,Z 539.458,A -85,B 0,C 180,E1 -13761.255,E2 -13761.255} C_VEL
LIN {X 0,Y 346.341,Z 544.388,A -85,B 0,C 180,E1 -13763.008,E2 -13763.008} C_VEL
LIN {X 0,Y 346.192,Z 547.706,A -85,B 0,C 180,E1 -13764.504,E2 -13764.504} C_VEL
LIN {X 0,Y 346.148,Z 550.929,A -85,B 0,C 180,E1 -13766.509,E2 -13766.509} C_VEL
LIN {X 0,Y 346.122,Z 553.122,A -85,B 0,C 180,E1 -13768.837,E2 -13768.837} C_VEL
LIN {X 0,Y 346.165,Z 553.601,A -85,B 0,C 180,E1 -13770.001,E2 -13770.001} C_VEL
LIN {X 0,Y 346.115,Z 553.659,A -85,B 0,C 180,E1 -13771.164,E2 -13771.164} C_VEL
LIN {X 0,Y 346.141,Z 552.627,A -85,B 0,C 180,E1 -13773.493,E2 -13773.493} C_VEL
LIN {X 0,Y 346.163,Z 551.512,A -85,B 0,C 180,E1 -13774.659,E2 -13774.659} C_VEL
LIN {X 0,Y 346.242,Z 549.754,A -85,B 0,C 180,E1 -13775.957,E2 -13775.957} C_VEL
LIN {X 0,Y 346.631,Z 545.599,A -85,B 0,C 180,E1 -13778.16,E2 -13778.16} C_VEL
LIN {X 0,Y 347.132,Z 541.081,A -85,B 0,C 180,E1 -13779.91,E2 -13779.91} C_VEL
LIN {X 0,Y 348.03,Z 534.263,A -85,B 0,C 180,E1 -13781.946,E2 -13781.946} C_VEL
LIN {X 0,Y 349.22,Z 526.884,A -85,B 0,C 180,E1 -13783.679,E2 -13783.679} C_VEL
LIN {X 0,Y 350.52,Z 518.368,A -85,B 0,C 180,E1 -13785.296,E2 -13785.296} C_VEL
LIN {X 0,Y 351.654,Z 509.333,A -85,B 0,C 180,E1 -13786.697,E2 -13786.697} C_VEL
LIN {X 0,Y 353.117,Z 499.063,A -85,B 0,C 180,E1 -13787.969,E2 -13787.969} C_VEL
LIN {X 0,Y 354.544,Z 487.697,A -85,B 0,C 180,E1 -13789.092,E2 -13789.092} C_VEL
LIN {X 0,Y 355.799,Z 475.869,A -85,B 0,C 180,E1 -13789.998,E2 -13789.998} C_VEL
LIN {X 0,Y 356.921,Z 463.528,A -85,B 0,C 180,E1 -13790.684,E2 -13790.684} C_VEL
LIN {X 0,Y 357.722,Z 449.846,A -85,B 0,C 180,E1 -13791.2,E2 -13791.2} C_VEL
LIN {X 0,Y 359.239,Z 376.498,A -85,B 0,C 180,E1 -13792.724,E2 -13792.724} C_VEL
LIN {X 0,Y 355.558,Z 356.071,A -85,B 0,C 180,E1 -13793.468,E2 -13793.468} C_VEL
LIN {X 0,Y 352.287,Z 340.609,A -85,B 0,C 180,E1 -13794.126,E2 -13794.126} C_VEL
LIN {X 0,Y 352.748,Z 335.549,A -85,B 0,C 180,E1 -13795.364,E2 -13795.364} C_VEL
LIN {X 0,Y 350.9,Z 325.138,A -85,B 0,C 180,E1 -13798.206,E2 -13798.206} C_VEL
LIN {X 0,Y 348.329,Z 314.5,A -85,B 0,C 180,E1 -13801.302,E2 -13801.302} C_VEL
LIN {X 0,Y 347.748,Z 312.169,A -85,B 0,C 180,E1 -13802.038,E2 -13802.038} C_VEL
LIN {X 0,Y 347.79,Z 312.165,A -85,B 0,C 180,E1 -13805.876,E2 -13805.876} C_VEL
LIN {X 0,Y 347.733,Z 312.17,A -85,B 0,C 180,E1 -13808.796,E2 -13808.796} C_VEL
LIN {X 0,Y 347.75,Z 312.166,A -85,B 0,C 180,E1 -13811.831,E2 -13811.831} C_VEL
LIN {X 0,Y 347.707,Z 312.173,A -85,B 0,C 180,E1 -13815.027,E2 -13815.027} C_VEL
LIN {X 0,Y 347.75,Z 312.166,A -85,B 0,C 180,E1 -13818.398,E2 -13818.398} C_VEL
LIN {X 0,Y 347.765,Z 312.16,A -85,B 0,C 180,E1 -13822.014,E2 -13822.014} C_VEL
LIN {X 0,Y 347.746,Z 312.165,A -85,B 0,C 180,E1 -13825.536,E2 -13825.536} C_VEL
LIN {X 0,Y 347.746,Z 312.161,A -85,B 0,C 180,E1 -13828.301,E2 -13828.301} C_VEL
LIN {X 0,Y 347.759,Z 312.163,A -85,B 0,C 180,E1 -13830.986,E2 -13830.986} C_VEL
LIN {X 0,Y 347.794,Z 312.159,A -85,B 0,C 180,E1 -13834.89,E2 -13834.89} C_VEL
LIN {X 0,Y 347.782,Z 312.16,A -85,B 0,C 180,E1 -13838.67,E2 -13838.67} C_VEL
LIN {X 0,Y 347.845,Z 312.15,A -85,B 0,C 180,E1 -13842.358,E2 -13842.358} C_VEL
LIN {X 0,Y 347.9,Z 312.144,A -85,B 0,C 180,E1 -13845.971,E2 -13845.971} C_VEL
LIN {X 0,Y 347.928,Z 312.143,A -85,B 0,C 180,E1 -13849.526,E2 -13849.526} C_VEL
LIN {X 0,Y 348.078,Z 312.119,A -85,B 0,C 180,E1 -13853.042,E2 -13853.042} C_VEL
LIN {X 0,Y 348.196,Z 312.106,A -85,B 0,C 180,E1 -13857.687,E2 -13857.687} C_VEL
LIN {X 0,Y 348.286,Z 312.093,A -85,B 0,C 180,E1 -13860,E2 -13860} C_VEL
LIN {X 0,Y 348.198,Z 312.111,A -85,B 0,C 180,E1 -13862.314,E2 -13862.314} C_VEL
LIN {X 0,Y 348.069,Z 312.125,A -85,B 0,C 180,E1 -13866.959,E2 -13866.959} C_VEL
LIN {X 0,Y 347.898,Z 312.147,A -85,B 0,C 180,E1 -13870.476,E2 -13870.476} C_VEL
LIN {X 0,Y 347.901,Z 312.142,A -85,B 0,C 180,E1 -13874.15,E2 -13874.15} C_VEL
LIN {X 0,Y 347.832,Z 312.15,A -85,B 0,C 180,E1 -13878.259,E2 -13878.259} C_VEL
LIN {X 0,Y 347.771,Z 312.157,A -85,B 0,C 180,E1 -13881.626,E2 -13881.626} C_VEL
LIN {X 0,Y 347.795,Z 312.156,A -85,B 0,C 180,E1 -13885.11,E2 -13885.11} C_VEL
LIN {X 0,Y 347.76,Z 312.161,A -85,B 0,C 180,E1 -13889.015,E2 -13889.015} C_VEL
LIN {X 0,Y 347.736,Z 312.169,A -85,B 0,C 180,E1 -13893.072,E2 -13893.072} C_VEL
LIN {X 0,Y 347.773,Z 312.164,A -85,B 0,C 180,E1 -13896.065,E2 -13896.065} C_VEL
LIN {X 0,Y 347.755,Z 312.167,A -85,B 0,C 180,E1 -13898.793,E2 -13898.793} C_VEL
LIN {X 0,Y 347.751,Z 312.167,A -85,B 0,C 180,E1 -13901.831,E2 -13901.831} C_VEL
LIN {X 0,Y 347.709,Z 312.174,A -85,B 0,C 180,E1 -13905.027,E2 -13905.027} C_VEL
LIN {X 0,Y 347.745,Z 312.172,A -85,B 0,C 180,E1 -13908.399,E2 -13908.399} C_VEL
LIN {X 0,Y 347.79,Z 312.252,A -85,B 0,C 180,E1 -13911.434,E2 -13911.434} C_VEL
LIN {X 0,Y 350.423,Z 323.575,A -85,B 0,C 180,E1 -13914.794,E2 -13914.794} C_VEL
LIN {X 0,Y 356.595,Z 338.146,A -85,B 0,C 180,E1 -13915.646,E2 -13915.646} C_VEL
LIN {X 0,Y 359.854,Z 352.944,A -85,B 0,C 180,E1 -13916.236,E2 -13916.236} C_VEL
LIN {X 0,Y 358.03,Z 431.045,A -85,B 0,C 180,E1 -13917.836,E2 -13917.836} C_VEL
LIN {X 0,Y 357.373,Z 443.647,A -85,B 0,C 180,E1 -13918.301,E2 -13918.301} C_VEL
LIN {X 0,Y 356.392,Z 456.259,A -85,B 0,C 180,E1 -13918.99,E2 -13918.99} C_VEL
LIN {X 0,Y 355.368,Z 468.054,A -85,B 0,C 180,E1 -13919.878,E2 -13919.878} C_VEL
LIN {X 0,Y 354.141,Z 479.077,A -85,B 0,C 180,E1 -13920.953,E2 -13920.953} C_VEL
LIN {X 0,Y 352.701,Z 489.636,A -85,B 0,C 180,E1 -13922.239,E2 -13922.239} C_VEL
LIN {X 0,Y 351.4,Z 498.509,A -85,B 0,C 180,E1 -13923.576,E2 -13923.576} C_VEL
LIN {X 0,Y 350.229,Z 506.63,A -85,B 0,C 180,E1 -13925.076,E2 -13925.076} C_VEL
LIN {X 0,Y 348.956,Z 514.465,A -85,B 0,C 180,E1 -13926.875,E2 -13926.875} C_VEL
LIN {X 0,Y 348.005,Z 520.708,A -85,B 0,C 180,E1 -13928.683,E2 -13928.683} C_VEL
LIN {X 0,Y 347.267,Z 525.607,A -85,B 0,C 180,E1 -13930.492,E2 -13930.492} C_VEL
LIN {X 0,Y 346.773,Z 529.323,A -85,B 0,C 180,E1 -13932.301,E2 -13932.301} C_VEL
LIN {X 0,Y 346.495,Z 531.221,A -85,B 0,C 180,E1 -13933.502,E2 -13933.502} C_VEL
LIN {X 0,Y 346.248,Z 532.627,A -85,B 0,C 180,E1 -13934.7,E2 -13934.7} C_VEL
LIN {X 0,Y 346.133,Z 534.191,A -85,B 0,C 180,E1 -13937.063,E2 -13937.063} C_VEL
LIN {X 0,Y 346.042,Z 534.374,A -85,B 0,C 180,E1 -13938.281,E2 -13938.281} C_VEL
LIN {X 0,Y 345.992,Z 534.112,A -85,B 0,C 180,E1 -13939.466,E2 -13939.466} C_VEL
LIN {X 0,Y 346.08,Z 532.415,A -85,B 0,C 180,E1 -13941.827,E2 -13941.827} C_VEL
LIN {X 0,Y 346.286,Z 529.372,A -85,B 0,C 180,E1 -13943.978,E2 -13943.978} C_VEL
LIN {X 0,Y 346.557,Z 525.301,A -85,B 0,C 180,E1 -13945.929,E2 -13945.929} C_VEL
LIN {X 0,Y 346.951,Z 520.475,A -85,B 0,C 180,E1 -13947.677,E2 -13947.677} C_VEL
LIN {X 0,Y 347.414,Z 514.404,A -85,B 0,C 180,E1 -13949.42,E2 -13949.42} C_VEL
LIN {X 0,Y 348.307,Z 506.836,A -85,B 0,C 180,E1 -13951.155,E2 -13951.155} C_VEL
LIN {X 0,Y 348.977,Z 499.135,A -85,B 0,C 180,E1 -13952.596,E2 -13952.596} C_VEL
LIN {X 0,Y 349.859,Z 489.727,A -85,B 0,C 180,E1 -13954.031,E2 -13954.031} C_VEL
LIN {X 0,Y 351.033,Z 479.242,A -85,B 0,C 180,E1 -13955.312,E2 -13955.312} C_VEL
LIN {X 0,Y 351.959,Z 467.637,A -85,B 0,C 180,E1 -13956.448,E2 -13956.448} C_VEL
LIN {X 0,Y 352.697,Z 455.298,A -85,B 0,C 180,E1 -13957.369,E2 -13957.369} C_VEL
LIN {X 0,Y 353.345,Z 442.294,A -85,B 0,C 180,E1 -13958.074,E2 -13958.074} C_VEL
LIN {X 0,Y 353.837,Z 429.38,A -85,B 0,C 180,E1 -13958.53,E2 -13958.53} C_VEL
LIN {X 0,Y 355.331,Z 350.262,A -85,B 0,C 180,E1 -13960.127,E2 -13960.127} C_VEL
LIN {X 0,Y 351.306,Z 327.437,A -85,B 0,C 180,E1 -13960.823,E2 -13960.823} C_VEL
LIN {X 0,Y 349.991,Z 323.162,A -85,B 0,C 180,E1 -13960.991,E2 -13960.991} C_VEL
LIN {X 0,Y 348.844,Z 316.873,A -85,B 0,C 180,E1 -13962.707,E2 -13962.707} C_VEL
LIN {X 0,Y 347.826,Z 315.159,A -85,B 0,C 180,E1 -13963.277,E2 -13963.277} C_VEL
LIN {X 0,Y 345.987,Z 314.055,A -85,B 0,C 180,E1 -13963.847,E2 -13963.847} C_VEL
LIN {X 0,Y 342.002,Z 313.131,A -85,B 0,C 180,E1 -13965.033,E2 -13965.033} C_VEL
LIN {X 0,Y 340.873,Z 313.038,A -85,B 0,C 180,E1 -13965.687,E2 -13965.687} C_VEL
LIN {X 0,Y 340.771,Z 313.034,A -85,B 0,C 180,E1 -13965.913,E2 -13965.913} C_VEL
LIN {X 0,Y 340.736,Z 313.038,A -85,B 0,C 180,E1 -13969.269,E2 -13969.269} C_VEL
LIN {X 0,Y 340.706,Z 313.041,A -85,B 0,C 180,E1 -13973.073,E2 -13973.073} C_VEL
LIN {X 0,Y 340.71,Z 313.042,A -85,B 0,C 180,E1 -13976.987,E2 -13976.987} C_VEL
LIN {X 0,Y 340.689,Z 313.044,A -85,B 0,C 180,E1 -13981.044,E2 -13981.044} C_VEL
LIN {X 0,Y 340.713,Z 313.041,A -85,B 0,C 180,E1 -13985.278,E2 -13985.278} C_VEL
LIN {X 0,Y 340.69,Z 313.047,A -85,B 0,C 180,E1 -13988.381,E2 -13988.381} C_VEL
LIN {X 0,Y 340.687,Z 313.044,A -85,B 0,C 180,E1 -13992.042,E2 -13992.042} C_VEL
LIN {X 0,Y 340.645,Z 313.049,A -85,B 0,C 180,E1 -13996.226,E2 -13996.226} C_VEL
LIN {X 0,Y 340.664,Z 313.049,A -85,B 0,C 180,E1 -13998.687,E2 -13998.687} C_VEL
LIN {X 0,Y 340.713,Z 313.041,A -85,B 0,C 180,E1 -14001.769,E2 -14001.769} C_VEL
LIN {X 0,Y 340.716,Z 313.042,A -85,B 0,C 180,E1 -14005.595,E2 -14005.595} C_VEL
LIN {X 0,Y 340.674,Z 313.048,A -85,B 0,C 180,E1 -14008.952,E2 -14008.952} C_VEL
LIN {X 0,Y 340.703,Z 313.043,A -85,B 0,C 180,E1 -14013.011,E2 -14013.011} C_VEL
LIN {X 0,Y 340.697,Z 313.043,A -85,B 0,C 180,E1 -14016.925,E2 -14016.925} C_VEL
LIN {X 0,Y 340.699,Z 313.042,A -85,B 0,C 180,E1 -14020.728,E2 -14020.728} C_VEL
LIN {X 0,Y 340.723,Z 313.04,A -85,B 0,C 180,E1 -14023.215,E2 -14023.215} C_VEL
LIN {X 0,Y 340.806,Z 313.028,A -85,B 0,C 180,E1 -14026.889,E2 -14026.889} C_VEL
LIN {X 0,Y 340.871,Z 313.023,A -85,B 0,C 180,E1 -14030.506,E2 -14030.506} C_VEL
LIN {X 0,Y 340.994,Z 313.005,A -85,B 0,C 180,E1 -14032.896,E2 -14032.896} C_VEL
LIN {X 0,Y 340.809,Z 313.027,A -85,B 0,C 180,E1 -14035.268,E2 -14035.268} C_VEL
LIN {X 0,Y 341.12,Z 312.99,A -85,B 0,C 180,E1 -14037.638,E2 -14037.638} C_VEL
LIN {X 0,Y 341.1,Z 312.992,A -85,B 0,C 180,E1 -14041.18,E2 -14041.18} C_VEL
LIN {X 0,Y 341.118,Z 312.996,A -85,B 0,C 180,E1 -14042.361,E2 -14042.361} C_VEL
LIN {X 0,Y 341.011,Z 313.004,A -85,B 0,C 180,E1 -14047.103,E2 -14047.103} C_VEL
LIN {X 0,Y 340.838,Z 313.031,A -85,B 0,C 180,E1 -14050.695,E2 -14050.695} C_VEL
LIN {X 0,Y 340.855,Z 313.024,A -85,B 0,C 180,E1 -14054.325,E2 -14054.325} C_VEL
LIN {X 0,Y 340.777,Z 313.034,A -85,B 0,C 180,E1 -14058.441,E2 -14058.441} C_VEL
LIN {X 0,Y 340.71,Z 313.041,A -85,B 0,C 180,E1 -14061.842,E2 -14061.842} C_VEL
LIN {X 0,Y 340.752,Z 313.037,A -85,B 0,C 180,E1 -14065.666,E2 -14065.666} C_VEL
LIN {X 0,Y 340.718,Z 313.039,A -85,B 0,C 180,E1 -14068.322,E2 -14068.322} C_VEL
LIN {X 0,Y 340.691,Z 313.047,A -85,B 0,C 180,E1 -14071.045,E2 -14071.045} C_VEL
LIN {X 0,Y 340.711,Z 313.045,A -85,B 0,C 180,E1 -14075.28,E2 -14075.28} C_VEL
LIN {X 0,Y 340.688,Z 313.044,A -85,B 0,C 180,E1 -14078.383,E2 -14078.383} C_VEL
LIN {X 0,Y 340.691,Z 313.045,A -85,B 0,C 180,E1 -14082.046,E2 -14082.046} C_VEL
LIN {X 0,Y 340.646,Z 313.051,A -85,B 0,C 180,E1 -14086.228,E2 -14086.228} C_VEL
LIN {X 0,Y 340.681,Z 313.049,A -85,B 0,C 180,E1 -14089.755,E2 -14089.755} C_VEL
LIN {X 0,Y 340.7,Z 313.042,A -85,B 0,C 180,E1 -14093.259,E2 -14093.259} C_VEL
LIN {X 0,Y 340.691,Z 313.05,A -85,B 0,C 180,E1 -14096.155,E2 -14096.155} C_VEL
LIN {X 0,Y 340.768,Z 313.04,A -85,B 0,C 180,E1 -14100.461,E2 -14100.461} C_VEL
LIN {X 0,Y 342.761,Z 323.12,A -85,B 0,C 180,E1 -14103.188,E2 -14103.188} C_VEL
LIN {X 0,Y 344.085,Z 331.054,A -85,B 0,C 180,E1 -14105.248,E2 -14105.248} C_VEL
LIN {X 0,Y 343.165,Z 341.003,A -85,B 0,C 180,E1 -14107.645,E2 -14107.645} C_VEL
LIN {X 0,Y 348.293,Z 376.808,A -85,B 0,C 180,E1 -14108.704,E2 -14108.704} C_VEL
LIN {X 0,Y 347.077,Z 449.289,A -85,B 0,C 180,E1 -14110.213,E2 -14110.213} C_VEL
LIN {X 0,Y 346.444,Z 462.603,A -85,B 0,C 180,E1 -14110.715,E2 -14110.715} C_VEL
LIN {X 0,Y 345.598,Z 474.804,A -85,B 0,C 180,E1 -14111.398,E2 -14111.398} C_VEL
LIN {X 0,Y 344.567,Z 487.106,A -85,B 0,C 180,E1 -14112.339,E2 -14112.339} C_VEL
LIN {X 0,Y 343.402,Z 498.74,A -85,B 0,C 180,E1 -14113.504,E2 -14113.504} C_VEL
LIN {X 0,Y 342.529,Z 509.233,A -85,B 0,C 180,E1 -14114.835,E2 -14114.835} C_VEL
LIN {X 0,Y 341.489,Z 518.628,A -85,B 0,C 180,E1 -14116.311,E2 -14116.311} C_VEL
LIN {X 0,Y 340.723,Z 526.349,A -85,B 0,C 180,E1 -14117.795,E2 -14117.795} C_VEL
LIN {X 0,Y 340.014,Z 533.902,A -85,B 0,C 180,E1 -14119.581,E2 -14119.581} C_VEL
LIN {X 0,Y 339.475,Z 540.867,A -85,B 0,C 180,E1 -14121.668,E2 -14121.668} C_VEL
LIN {X 0,Y 339.231,Z 545.448,A -85,B 0,C 180,E1 -14123.458,E2 -14123.458} C_VEL
LIN {X 0,Y 339.098,Z 548.92,A -85,B 0,C 180,E1 -14125.246,E2 -14125.246} C_VEL
LIN {X 0,Y 339.074,Z 550.648,A -85,B 0,C 180,E1 -14126.436,E2 -14126.436} C_VEL
LIN {X 0,Y 339.024,Z 552.877,A -85,B 0,C 180,E1 -14128.813,E2 -14128.813} C_VEL
LIN {X 0,Y 339.068,Z 553.391,A -85,B 0,C 180,E1 -14130.001,E2 -14130.001} C_VEL
LIN {X 0,Y 339.017,Z 553.469,A -85,B 0,C 180,E1 -14131.189,E2 -14131.189} C_VEL
LIN {X 0,Y 339.065,Z 552.474,A -85,B 0,C 180,E1 -14133.566,E2 -14133.566} C_VEL
LIN {X 0,Y 339.068,Z 551.391,A -85,B 0,C 180,E1 -14134.757,E2 -14134.757} C_VEL
LIN {X 0,Y 339.141,Z 549.861,A -85,B 0,C 180,E1 -14135.948,E2 -14135.948} C_VEL
LIN {X 0,Y 339.421,Z 546.796,A -85,B 0,C 180,E1 -14137.736,E2 -14137.736} C_VEL
LIN {X 0,Y 339.93,Z 542.693,A -85,B 0,C 180,E1 -14139.521,E2 -14139.521} C_VEL
LIN {X 0,Y 340.777,Z 536.433,A -85,B 0,C 180,E1 -14141.601,E2 -14141.601} C_VEL
LIN {X 0,Y 341.89,Z 529.638,A -85,B 0,C 180,E1 -14143.372,E2 -14143.372} C_VEL
LIN {X 0,Y 343.247,Z 521.202,A -85,B 0,C 180,E1 -14145.134,E2 -14145.134} C_VEL
LIN {X 0,Y 344.444,Z 512.55,A -85,B 0,C 180,E1 -14146.599,E2 -14146.599} C_VEL
LIN {X 0,Y 345.881,Z 503.083,A -85,B 0,C 180,E1 -14147.899,E2 -14147.899} C_VEL
LIN {X 0,Y 347.291,Z 492.779,A -85,B 0,C 180,E1 -14149.046,E2 -14149.046} C_VEL
LIN {X 0,Y 348.731,Z 481.495,A -85,B 0,C 180,E1 -14150.036,E2 -14150.036} C_VEL
LIN {X 0,Y 349.838,Z 469.99,A -85,B 0,C 180,E1 -14150.814,E2 -14150.814} C_VEL
LIN {X 0,Y 350.911,Z 456.779,A -85,B 0,C 180,E1 -14151.44,E2 -14151.44} C_VEL
LIN {X 0,Y 351.508,Z 444.005,A -85,B 0,C 180,E1 -14151.825,E2 -14151.825} C_VEL
LIN {X 0,Y 352.876,Z 377.533,A -85,B 0,C 180,E1 -14153.207,E2 -14153.207} C_VEL
LIN {X 0,Y 349.388,Z 358.07,A -85,B 0,C 180,E1 -14153.937,E2 -14153.937} C_VEL
LIN {X 0,Y 345.598,Z 340.424,A -85,B 0,C 180,E1 -14154.703,E2 -14154.703} C_VEL
LIN {X 0,Y 345.894,Z 337.018,A -85,B 0,C 180,E1 -14155.557,E2 -14155.557} C_VEL
LIN {X 0,Y 344.403,Z 328.247,A -85,B 0,C 180,E1 -14157.992,E2 -14157.992} C_VEL
LIN {X 0,Y 341.734,Z 317.125,A -85,B 0,C 180,E1 -14161.285,E2 -14161.285} C_VEL
LIN {X 0,Y 340.717,Z 313.044,A -85,B 0,C 180,E1 -14162.608,E2 -14162.608} C_VEL
LIN {X 0,Y 340.72,Z 313.048,A -85,B 0,C 180,E1 -14165.279,E2 -14165.279} C_VEL
LIN {X 0,Y 340.697,Z 313.049,A -85,B 0,C 180,E1 -14168.383,E2 -14168.383} C_VEL
LIN {X 0,Y 340.699,Z 313.045,A -85,B 0,C 180,E1 -14172.045,E2 -14172.045} C_VEL
LIN {X 0,Y 340.654,Z 313.05,A -85,B 0,C 180,E1 -14176.227,E2 -14176.227} C_VEL
LIN {X 0,Y 340.677,Z 313.046,A -85,B 0,C 180,E1 -14179.756,E2 -14179.756} C_VEL
LIN {X 0,Y 340.704,Z 313.044,A -85,B 0,C 180,E1 -14183.258,E2 -14183.258} C_VEL
LIN {X 0,Y 340.694,Z 313.044,A -85,B 0,C 180,E1 -14186.154,E2 -14186.154} C_VEL
LIN {X 0,Y 340.733,Z 313.04,A -85,B 0,C 180,E1 -14190.329,E2 -14190.329} C_VEL
LIN {X 0,Y 340.746,Z 313.038,A -85,B 0,C 180,E1 -14194.334,E2 -14194.334} C_VEL
LIN {X 0,Y 340.743,Z 313.036,A -85,B 0,C 180,E1 -14198.207,E2 -14198.207} C_VEL
LIN {X 0,Y 340.794,Z 313.029,A -85,B 0,C 180,E1 -14201.981,E2 -14201.981} C_VEL
LIN {X 0,Y 340.871,Z 313.022,A -85,B 0,C 180,E1 -14205.705,E2 -14205.705} C_VEL
LIN {X 0,Y 340.871,Z 313.02,A -85,B 0,C 180,E1 -14209.306,E2 -14209.306} C_VEL
LIN {X 0,Y 341.047,Z 312.994,A -85,B 0,C 180,E1 -14212.898,E2 -14212.898} C_VEL
LIN {X 0,Y 341.133,Z 312.985,A -85,B 0,C 180,E1 -14217.639,E2 -14217.639} C_VEL
LIN {X 0,Y 341.238,Z 312.97,A -85,B 0,C 180,E1 -14220,E2 -14220} C_VEL
LIN {X 0,Y 341.159,Z 312.988,A -85,B 0,C 180,E1 -14222.362,E2 -14222.362} C_VEL
LIN {X 0,Y 341.018,Z 313.003,A -85,B 0,C 180,E1 -14227.103,E2 -14227.103} C_VEL
LIN {X 0,Y 340.85,Z 313.028,A -85,B 0,C 180,E1 -14230.695,E2 -14230.695} C_VEL
LIN {X 0,Y 340.866,Z 313.019,A -85,B 0,C 180,E1 -14234.325,E2 -14234.325} C_VEL
LIN {X 0,Y 340.789,Z 313.028,A -85,B 0,C 180,E1 -14238.441,E2 -14238.441} C_VEL
LIN {X 0,Y 340.721,Z 313.035,A -85,B 0,C 180,E1 -14241.842,E2 -14241.842} C_VEL
LIN {X 0,Y 340.747,Z 313.035,A -85,B 0,C 180,E1 -14245.667,E2 -14245.667} C_VEL
LIN {X 0,Y 340.735,Z 313.04,A -85,B 0,C 180,E1 -14249.672,E2 -14249.672} C_VEL
LIN {X 0,Y 340.696,Z 313.043,A -85,B 0,C 180,E1 -14253.847,E2 -14253.847} C_VEL
LIN {X 0,Y 340.707,Z 313.044,A -85,B 0,C 180,E1 -14256.742,E2 -14256.742} C_VEL
LIN {X 0,Y 340.689,Z 313.047,A -85,B 0,C 180,E1 -14260.246,E2 -14260.246} C_VEL
LIN {X 0,Y 340.655,Z 313.051,A -85,B 0,C 180,E1 -14263.773,E2 -14263.773} C_VEL
LIN {X 0,Y 340.697,Z 313.049,A -85,B 0,C 180,E1 -14267.956,E2 -14267.956} C_VEL
LIN {X 0,Y 340.718,Z 313.132,A -85,B 0,C 180,E1 -14270.898,E2 -14270.898} C_VEL
LIN {X 0,Y 343.256,Z 323.666,A -85,B 0,C 180,E1 -14274.155,E2 -14274.155} C_VEL
LIN {X 0,Y 350.625,Z 340.857,A -85,B 0,C 180,E1 -14275.205,E2 -14275.205} C_VEL
LIN {X 0,Y 353.442,Z 353.331,A -85,B 0,C 180,E1 -14275.725,E2 -14275.725} C_VEL
LIN {X 0,Y 351.644,Z 430.778,A -85,B 0,C 180,E1 -14277.341,E2 -14277.341} C_VEL
LIN {X 0,Y 350.94,Z 443.277,A -85,B 0,C 180,E1 -14277.799,E2 -14277.799} C_VEL
LIN {X 0,Y 349.911,Z 456.328,A -85,B 0,C 180,E1 -14278.519,E2 -14278.519} C_VEL
LIN {X 0,Y 348.83,Z 468.154,A -85,B 0,C 180,E1 -14279.421,E2 -14279.421} C_VEL
LIN {X 0,Y 347.527,Z 479.299,A -85,B 0,C 180,E1 -14280.525,E2 -14280.525} C_VEL
LIN {X 0,Y 346.049,Z 489.771,A -85,B 0,C 180,E1 -14281.823,E2 -14281.823} C_VEL
LIN {X 0,Y 344.524,Z 499.558,A -85,B 0,C 180,E1 -14283.334,E2 -14283.334} C_VEL
LIN {X 0,Y 343.302,Z 507.499,A -85,B 0,C 180,E1 -14284.862,E2 -14284.862} C_VEL
LIN {X 0,Y 341.993,Z 515.203,A -85,B 0,C 180,E1 -14286.697,E2 -14286.697} C_VEL
LIN {X 0,Y 341.161,Z 520.417,A -85,B 0,C 180,E1 -14288.234,E2 -14288.234} C_VEL
LIN {X 0,Y 340.338,Z 525.42,A -85,B 0,C 180,E1 -14290.078,E2 -14290.078} C_VEL
LIN {X 0,Y 339.736,Z 529.545,A -85,B 0,C 180,E1 -14292.1,E2 -14292.1} C_VEL
LIN {X 0,Y 339.209,Z 532.677,A -85,B 0,C 180,E1 -14294.374,E2 -14294.374} C_VEL
LIN {X 0,Y 339.089,Z 533.708,A -85,B 0,C 180,E1 -14295.598,E2 -14295.598} C_VEL
LIN {X 0,Y 339.043,Z 534.4,A -85,B 0,C 180,E1 -14296.974,E2 -14296.974} C_VEL
LIN {X 0,Y 338.921,Z 534.377,A -85,B 0,C 180,E1 -14299.243,E2 -14299.243} C_VEL
LIN {X 0,Y 338.97,Z 532.767,A -85,B 0,C 180,E1 -14301.654,E2 -14301.654} C_VEL
LIN {X 0,Y 339.09,Z 531.364,A -85,B 0,C 180,E1 -14302.856,E2 -14302.856} C_VEL
LIN {X 0,Y 339.315,Z 528.422,A -85,B 0,C 180,E1 -14304.651,E2 -14304.651} C_VEL
LIN {X 0,Y 339.551,Z 524.453,A -85,B 0,C 180,E1 -14306.439,E2 -14306.439} C_VEL
LIN {X 0,Y 340.052,Z 518.341,A -85,B 0,C 180,E1 -14308.519,E2 -14308.519} C_VEL
LIN {X 0,Y 340.709,Z 511.675,A -85,B 0,C 180,E1 -14310.295,E2 -14310.295} C_VEL
LIN {X 0,Y 341.644,Z 503.401,A -85,B 0,C 180,E1 -14312.062,E2 -14312.062} C_VEL
LIN {X 0,Y 342.371,Z 494.939,A -85,B 0,C 180,E1 -14313.53,E2 -14313.53} C_VEL
LIN {X 0,Y 343.563,Z 484.44,A -85,B 0,C 180,E1 -14314.987,E2 -14314.987} C_VEL
LIN {X 0,Y 344.596,Z 474.051,A -85,B 0,C 180,E1 -14316.146,E2 -14316.146} C_VEL
LIN {X 0,Y 345.433,Z 462.694,A -85,B 0,C 180,E1 -14317.158,E2 -14317.158} C_VEL
LIN {X 0,Y 346.104,Z 450.99,A -85,B 0,C 180,E1 -14317.951,E2 -14317.951} C_VEL
LIN {X 0,Y 346.74,Z 437.479,A -85,B 0,C 180,E1 -14318.596,E2 -14318.596} C_VEL
LIN {X 0,Y 347.219,Z 425.361,A -85,B 0,C 180,E1 -14318.951,E2 -14318.951} C_VEL
LIN {X 0,Y 348.549,Z 351.08,A -85,B 0,C 180,E1 -14320.469,E2 -14320.469} C_VEL
LIN {X 0,Y 344.676,Z 329.214,A -85,B 0,C 180,E1 -14321.154,E2 -14321.154} C_VEL
LIN {X 0,Y 342.83,Z 323.338,A -85,B 0,C 180,E1 -14321.399,E2 -14321.399} C_VEL
LIN {X 0,Y 340.865,Z 313.027,A -85,B 0,C 180,E1 -14324.324,E2 -14324.324} C_VEL
LIN {X 0,Y 340.771,Z 313.034,A -85,B 0,C 180,E1 -14325.913,E2 -14325.913} C_VEL
LIN {X 0,Y 340.068,Z 313.122,A -85,B 0,C 180,E1 -14326.899,E2 -14326.899} C_VEL
LIN {X 0,Y 337.206,Z 313.48,A -85,B 0,C 180,E1 -14328.503,E2 -14328.503} C_VEL
LIN {X 0,Y 334.794,Z 313.782,A -85,B 0,C 180,E1 -14329.802,E2 -14329.802} C_VEL
LIN {X 0,Y 333.748,Z 313.91,A -85,B 0,C 180,E1 -14330.807,E2 -14330.807} C_VEL
LIN {X 0,Y 333.656,Z 313.92,A -85,B 0,C 180,E1 -14331.148,E2 -14331.148} C_VEL
LIN {X 0,Y 333.659,Z 313.92,A -85,B 0,C 180,E1 -14335.077,E2 -14335.077} C_VEL
LIN {X 0,Y 333.629,Z 313.924,A -85,B 0,C 180,E1 -14338.979,E2 -14338.979} C_VEL
LIN {X 0,Y 333.641,Z 313.927,A -85,B 0,C 180,E1 -14342.585,E2 -14342.585} C_VEL
LIN {X 0,Y 333.671,Z 313.919,A -85,B 0,C 180,E1 -14346.138,E2 -14346.138} C_VEL
LIN {X 0,Y 333.617,Z 313.926,A -85,B 0,C 180,E1 -14349.195,E2 -14349.195} C_VEL
LIN {X 0,Y 333.622,Z 313.926,A -85,B 0,C 180,E1 -14352.497,E2 -14352.497} C_VEL
LIN {X 0,Y 333.589,Z 313.927,A -85,B 0,C 180,E1 -14355.953,E2 -14355.953} C_VEL
LIN {X 0,Y 333.597,Z 313.93,A -85,B 0,C 180,E1 -14359.323,E2 -14359.323} C_VEL
LIN {X 0,Y 333.656,Z 313.925,A -85,B 0,C 180,E1 -14363.168,E2 -14363.168} C_VEL
LIN {X 0,Y 333.667,Z 313.922,A -85,B 0,C 180,E1 -14365.34,E2 -14365.34} C_VEL
LIN {X 0,Y 333.613,Z 313.925,A -85,B 0,C 180,E1 -14368.22,E2 -14368.22} C_VEL
LIN {X 0,Y 333.616,Z 313.927,A -85,B 0,C 180,E1 -14371.018,E2 -14371.018} C_VEL
LIN {X 0,Y 333.651,Z 313.919,A -85,B 0,C 180,E1 -14374.921,E2 -14374.921} C_VEL
LIN {X 0,Y 333.646,Z 313.922,A -85,B 0,C 180,E1 -14379.017,E2 -14379.017} C_VEL
LIN {X 0,Y 333.704,Z 313.918,A -85,B 0,C 180,E1 -14381.584,E2 -14381.584} C_VEL
LIN {X 0,Y 333.751,Z 313.909,A -85,B 0,C 180,E1 -14385.61,E2 -14385.61} C_VEL
LIN {X 0,Y 333.8,Z 313.901,A -85,B 0,C 180,E1 -14389.077,E2 -14389.077} C_VEL
LIN {X 0,Y 333.949,Z 313.883,A -85,B 0,C 180,E1 -14392.746,E2 -14392.746} C_VEL
LIN {X 0,Y 333.775,Z 313.902,A -85,B 0,C 180,E1 -14395.168,E2 -14395.168} C_VEL
LIN {X 0,Y 334.061,Z 313.869,A -85,B 0,C 180,E1 -14397.588,E2 -14397.588} C_VEL
LIN {X 0,Y 334.069,Z 313.868,A -85,B 0,C 180,E1 -14401.205,E2 -14401.205} C_VEL
LIN {X 0,Y 333.798,Z 313.901,A -85,B 0,C 180,E1 -14403.621,E2 -14403.621} C_VEL
LIN {X 0,Y 333.99,Z 313.878,A -85,B 0,C 180,E1 -14406.039,E2 -14406.039} C_VEL
LIN {X 0,Y 333.811,Z 313.9,A -85,B 0,C 180,E1 -14409.696,E2 -14409.696} C_VEL
LIN {X 0,Y 333.788,Z 313.903,A -85,B 0,C 180,E1 -14413.392,E2 -14413.392} C_VEL
LIN {X 0,Y 333.711,Z 313.916,A -85,B 0,C 180,E1 -14417.148,E2 -14417.148} C_VEL
LIN {X 0,Y 333.677,Z 313.917,A -85,B 0,C 180,E1 -14419.694,E2 -14419.694} C_VEL
LIN {X 0,Y 333.66,Z 313.92,A -85,B 0,C 180,E1 -14423.591,E2 -14423.591} C_VEL
LIN {X 0,Y 333.694,Z 313.915,A -85,B 0,C 180,E1 -14426.25,E2 -14426.25} C_VEL
LIN {X 0,Y 333.682,Z 313.919,A -85,B 0,C 180,E1 -14428.975,E2 -14428.975} C_VEL
LIN {X 0,Y 333.637,Z 313.922,A -85,B 0,C 180,E1 -14432.588,E2 -14432.588} C_VEL
LIN {X 0,Y 333.668,Z 313.919,A -85,B 0,C 180,E1 -14436.14,E2 -14436.14} C_VEL
LIN {X 0,Y 333.626,Z 313.926,A -85,B 0,C 180,E1 -14439.195,E2 -14439.195} C_VEL
LIN {X 0,Y 333.625,Z 313.923,A -85,B 0,C 180,E1 -14442.5,E2 -14442.5} C_VEL
LIN {X 0,Y 333.591,Z 313.933,A -85,B 0,C 180,E1 -14445.956,E2 -14445.956} C_VEL
LIN {X 0,Y 333.641,Z 313.923,A -85,B 0,C 180,E1 -14449.317,E2 -14449.317} C_VEL
LIN {X 0,Y 333.661,Z 313.919,A -85,B 0,C 180,E1 -14453.169,E2 -14453.169} C_VEL
LIN {X 0,Y 333.635,Z 313.924,A -85,B 0,C 180,E1 -14456.793,E2 -14456.793} C_VEL
LIN {X 0,Y 333.729,Z 313.92,A -85,B 0,C 180,E1 -14460.183,E2 -14460.183} C_VEL
LIN {X 0,Y 335.708,Z 323.864,A -85,B 0,C 180,E1 -14462.915,E2 -14462.915} C_VEL
LIN {X 0,Y 337.088,Z 331.808,A -85,B 0,C 180,E1 -14465.028,E2 -14465.028} C_VEL
LIN {X 0,Y 336.278,Z 340.842,A -85,B 0,C 180,E1 -14467.255,E2 -14467.255} C_VEL
LIN {X 0,Y 341.519,Z 378.248,A -85,B 0,C 180,E1 -14468.373,E2 -14468.373} C_VEL
LIN {X 0,Y 340.28,Z 449.15,A -85,B 0,C 180,E1 -14469.88,E2 -14469.88} C_VEL
LIN {X 0,Y 339.62,Z 462.442,A -85,B 0,C 180,E1 -14470.391,E2 -14470.391} C_VEL
LIN {X 0,Y 338.746,Z 474.633,A -85,B 0,C 180,E1 -14471.086,E2 -14471.086} C_VEL
LIN {X 0,Y 337.794,Z 486.124,A -85,B 0,C 180,E1 -14471.973,E2 -14471.973} C_VEL
LIN {X 0,Y 336.584,Z 497.91,A -85,B 0,C 180,E1 -14473.16,E2 -14473.16} C_VEL
LIN {X 0,Y 335.595,Z 507.954,A -85,B 0,C 180,E1 -14474.436,E2 -14474.436} C_VEL
LIN {X 0,Y 334.774,Z 516.251,A -85,B 0,C 180,E1 -14475.72,E2 -14475.72} C_VEL
LIN {X 0,Y 333.888,Z 524.358,A -85,B 0,C 180,E1 -14477.232,E2 -14477.232} C_VEL
LIN {X 0,Y 333.06,Z 532.296,A -85,B 0,C 180,E1 -14479.053,E2 -14479.053} C_VEL
LIN {X 0,Y 332.547,Z 538.626,A -85,B 0,C 180,E1 -14480.881,E2 -14480.881} C_VEL
LIN {X 0,Y 332.194,Z 543.65,A -85,B 0,C 180,E1 -14482.708,E2 -14482.708} C_VEL
LIN {X 0,Y 332.029,Z 546.868,A -85,B 0,C 180,E1 -14484.178,E2 -14484.178} C_VEL
LIN {X 0,Y 332,Z 550.361,A -85,B 0,C 180,E1 -14486.36,E2 -14486.36} C_VEL
LIN {X 0,Y 331.929,Z 552.629,A -85,B 0,C 180,E1 -14488.788,E2 -14488.788} C_VEL
LIN {X 0,Y 331.971,Z 553.173,A -85,B 0,C 180,E1 -14490.001,E2 -14490.001} C_VEL
LIN {X 0,Y 331.922,Z 553.28,A -85,B 0,C 180,E1 -14491.214,E2 -14491.214} C_VEL
LIN {X 0,Y 331.969,Z 552.323,A -85,B 0,C 180,E1 -14493.642,E2 -14493.642} C_VEL
LIN {X 0,Y 332.062,Z 550.052,A -85,B 0,C 180,E1 -14495.878,E2 -14495.878} C_VEL
LIN {X 0,Y 332.38,Z 546.747,A -85,B 0,C 180,E1 -14497.9,E2 -14497.9} C_VEL
LIN {X 0,Y 332.89,Z 542.688,A -85,B 0,C 180,E1 -14499.724,E2 -14499.724} C_VEL
LIN {X 0,Y 333.798,Z 536.477,A -85,B 0,C 180,E1 -14501.847,E2 -14501.847} C_VEL
LIN {X 0,Y 334.981,Z 529.736,A -85,B 0,C 180,E1 -14503.653,E2 -14503.653} C_VEL
LIN {X 0,Y 336.398,Z 521.39,A -85,B 0,C 180,E1 -14505.449,E2 -14505.449} C_VEL
LIN {X 0,Y 337.65,Z 512.827,A -85,B 0,C 180,E1 -14506.943,E2 -14506.943} C_VEL
LIN {X 0,Y 339.153,Z 503.462,A -85,B 0,C 180,E1 -14508.266,E2 -14508.266} C_VEL
LIN {X 0,Y 340.622,Z 493.287,A -85,B 0,C 180,E1 -14509.434,E2 -14509.434} C_VEL
LIN {X 0,Y 342.096,Z 482.18,A -85,B 0,C 180,E1 -14510.442,E2 -14510.442} C_VEL
LIN {X 0,Y 343.238,Z 470.98,A -85,B 0,C 180,E1 -14511.234,E2 -14511.234} C_VEL
LIN {X 0,Y 344.402,Z 458.415,A -85,B 0,C 180,E1 -14511.865,E2 -14511.865} C_VEL
LIN {X 0,Y 345.051,Z 445.354,A -85,B 0,C 180,E1 -14512.294,E2 -14512.294} C_VEL
LIN {X 0,Y 346.536,Z 378.48,A -85,B 0,C 180,E1 -14513.712,E2 -14513.712} C_VEL
LIN {X 0,Y 343.087,Z 359.332,A -85,B 0,C 180,E1 -14514.454,E2 -14514.454} C_VEL
LIN {X 0,Y 339.001,Z 340.187,A -85,B 0,C 180,E1 -14515.314,E2 -14515.314} C_VEL
LIN {X 0,Y 338.731,Z 336.647,A -85,B 0,C 180,E1 -14516.275,E2 -14516.275} C_VEL
LIN {X 0,Y 337.003,Z 327.722,A -85,B 0,C 180,E1 -14518.85,E2 -14518.85} C_VEL
LIN {X 0,Y 334.41,Z 316.911,A -85,B 0,C 180,E1 -14522.164,E2 -14522.164} C_VEL
LIN {X 0,Y 333.665,Z 313.926,A -85,B 0,C 180,E1 -14523.161,E2 -14523.161} C_VEL
LIN {X 0,Y 333.665,Z 313.925,A -85,B 0,C 180,E1 -14526.832,E2 -14526.832} C_VEL
LIN {X 0,Y 333.645,Z 313.924,A -85,B 0,C 180,E1 -14530.768,E2 -14530.768} C_VEL
LIN {X 0,Y 333.595,Z 313.93,A -85,B 0,C 180,E1 -14534.251,E2 -14534.251} C_VEL
LIN {X 0,Y 333.643,Z 313.924,A -85,B 0,C 180,E1 -14537.619,E2 -14537.619} C_VEL
LIN {X 0,Y 333.641,Z 313.919,A -85,B 0,C 180,E1 -14541.205,E2 -14541.205} C_VEL
LIN {X 0,Y 333.677,Z 313.918,A -85,B 0,C 180,E1 -14543.861,E2 -14543.861} C_VEL
LIN {X 0,Y 333.645,Z 313.918,A -85,B 0,C 180,E1 -14547.413,E2 -14547.413} C_VEL
LIN {X 0,Y 333.672,Z 313.917,A -85,B 0,C 180,E1 -14551.024,E2 -14551.024} C_VEL
LIN {X 0,Y 333.715,Z 313.911,A -85,B 0,C 180,E1 -14555.09,E2 -14555.09} C_VEL
LIN {X 0,Y 333.672,Z 313.916,A -85,B 0,C 180,E1 -14559.019,E2 -14559.019} C_VEL
LIN {X 0,Y 333.742,Z 313.911,A -85,B 0,C 180,E1 -14561.587,E2 -14561.587} C_VEL
LIN {X 0,Y 333.81,Z 313.903,A -85,B 0,C 180,E1 -14565.577,E2 -14565.577} C_VEL
LIN {X 0,Y 333.834,Z 313.895,A -85,B 0,C 180,E1 -14569.078,E2 -14569.078} C_VEL
LIN {X 0,Y 333.994,Z 313.873,A -85,B 0,C 180,E1 -14572.747,E2 -14572.747} C_VEL
LIN {X 0,Y 333.796,Z 313.898,A -85,B 0,C 180,E1 -14575.169,E2 -14575.169} C_VEL
LIN {X 0,Y 334.074,Z 313.864,A -85,B 0,C 180,E1 -14577.589,E2 -14577.589} C_VEL
LIN {X 0,Y 334.19,Z 313.848,A -85,B 0,C 180,E1 -14580,E2 -14580} C_VEL
LIN {X 0,Y 334.096,Z 313.867,A -85,B 0,C 180,E1 -14582.411,E2 -14582.411} C_VEL
LIN {X 0,Y 333.97,Z 313.877,A -85,B 0,C 180,E1 -14586.513,E2 -14586.513} C_VEL
LIN {X 0,Y 333.822,Z 313.893,A -85,B 0,C 180,E1 -14589.697,E2 -14589.697} C_VEL
LIN {X 0,Y 333.799,Z 313.896,A -85,B 0,C 180,E1 -14593.392,E2 -14593.392} C_VEL
LIN {X 0,Y 333.721,Z 313.907,A -85,B 0,C 180,E1 -14597.148,E2 -14597.148} C_VEL
LIN {X 0,Y 333.692,Z 313.916,A -85,B 0,C 180,E1 -14599.693,E2 -14599.693} C_VEL
LIN {X 0,Y 333.671,Z 313.918,A -85,B 0,C 180,E1 -14603.59,E2 -14603.59} C_VEL
LIN {X 0,Y 333.678,Z 313.915,A -85,B 0,C 180,E1 -14606.252,E2 -14606.252} C_VEL
LIN {X 0,Y 333.663,Z 313.919,A -85,B 0,C 180,E1 -14610.366,E2 -14610.366} C_VEL
LIN {X 0,Y 333.64,Z 313.926,A -85,B 0,C 180,E1 -14613.208,E2 -14613.208} C_VEL
LIN {X 0,Y 333.679,Z 313.92,A -85,B 0,C 180,E1 -14616.139,E2 -14616.139} C_VEL
LIN {X 0,Y 333.649,Z 313.925,A -85,B 0,C 180,E1 -14619.193,E2 -14619.193} C_VEL
LIN {X 0,Y 333.635,Z 313.926,A -85,B 0,C 180,E1 -14622.5,E2 -14622.5} C_VEL
LIN {X 0,Y 333.599,Z 313.931,A -85,B 0,C 180,E1 -14625.955,E2 -14625.955} C_VEL
LIN {X 0,Y 333.606,Z 313.926,A -85,B 0,C 180,E1 -14629.324,E2 -14629.324} C_VEL
LIN {X 0,Y 333.647,Z 313.956,A -85,B 0,C 180,E1 -14630.319,E2 -14630.319} C_VEL
LIN {X 0,Y 336.042,Z 323.896,A -85,B 0,C 180,E1 -14633.481,E2 -14633.481} C_VEL
LIN {X 0,Y 344.255,Z 342.412,A -85,B 0,C 180,E1 -14634.684,E2 -14634.684} C_VEL
LIN {X 0,Y 346.825,Z 352.903,A -85,B 0,C 180,E1 -14635.153,E2 -14635.153} C_VEL
LIN {X 0,Y 347.144,Z 356.051,A -85,B 0,C 180,E1 -14635.253,E2 -14635.253} C_VEL
LIN {X 0,Y 345.179,Z 432.002,A -85,B 0,C 180,E1 -14636.869,E2 -14636.869} C_VEL
LIN {X 0,Y 344.497,Z 443.773,A -85,B 0,C 180,E1 -14637.317,E2 -14637.317} C_VEL
LIN {X 0,Y 343.453,Z 456.454,A -85,B 0,C 180,E1 -14638.029,E2 -14638.029} C_VEL
LIN {X 0,Y 342.317,Z 468.295,A -85,B 0,C 180,E1 -14638.946,E2 -14638.946} C_VEL
LIN {X 0,Y 340.951,Z 479.559,A -85,B 0,C 180,E1 -14640.083,E2 -14640.083} C_VEL
LIN {X 0,Y 339.406,Z 489.921,A -85,B 0,C 180,E1 -14641.389,E2 -14641.389} C_VEL
LIN {X 0,Y 337.968,Z 498.806,A -85,B 0,C 180,E1 -14642.774,E2 -14642.774} C_VEL
LIN {X 0,Y 336.633,Z 506.939,A -85,B 0,C 180,E1 -14644.328,E2 -14644.328} C_VEL
LIN {X 0,Y 335.199,Z 514.792,A -85,B 0,C 180,E1 -14646.195,E2 -14646.195} C_VEL
LIN {X 0,Y 334.349,Z 520.125,A -85,B 0,C 180,E1 -14647.767,E2 -14647.767} C_VEL
LIN {X 0,Y 333.425,Z 525.234,A -85,B 0,C 180,E1 -14649.647,E2 -14649.647} C_VEL
LIN {X 0,Y 332.722,Z 529.787,A -85,B 0,C 180,E1 -14651.903,E2 -14651.903} C_VEL
LIN {X 0,Y 332.178,Z 532.709,A -85,B 0,C 180,E1 -14654.035,E2 -14654.035} C_VEL
LIN {X 0,Y 332.035,Z 533.802,A -85,B 0,C 180,E1 -14655.285,E2 -14655.285} C_VEL
LIN {X 0,Y 331.962,Z 534.607,A -85,B 0,C 180,E1 -14656.876,E2 -14656.876} C_VEL
LIN {X 0,Y 331.827,Z 534.638,A -85,B 0,C 180,E1 -14659.01,E2 -14659.01} C_VEL
LIN {X 0,Y 331.876,Z 533.116,A -85,B 0,C 180,E1 -14661.474,E2 -14661.474} C_VEL
LIN {X 0,Y 331.967,Z 531.763,A -85,B 0,C 180,E1 -14662.701,E2 -14662.701} C_VEL
LIN {X 0,Y 332.16,Z 529.222,A -85,B 0,C 180,E1 -14664.356,E2 -14664.356} C_VEL
LIN {X 0,Y 332.446,Z 525.028,A -85,B 0,C 180,E1 -14666.363,E2 -14666.363} C_VEL
LIN {X 0,Y 332.908,Z 520.02,A -85,B 0,C 180,E1 -14668.184,E2 -14668.184} C_VEL
LIN {X 0,Y 333.47,Z 513.742,A -85,B 0,C 180,E1 -14669.999,E2 -14669.999} C_VEL
LIN {X 0,Y 334.412,Z 505.861,A -85,B 0,C 180,E1 -14671.806,E2 -14671.806} C_VEL
LIN {X 0,Y 335.156,Z 497.869,A -85,B 0,C 180,E1 -14673.305,E2 -14673.305} C_VEL
LIN {X 0,Y 336.149,Z 489.158,A -85,B 0,C 180,E1 -14674.646,E2 -14674.646} C_VEL
LIN {X 0,Y 337.344,Z 478.488,A -85,B 0,C 180,E1 -14675.978,E2 -14675.978} C_VEL
LIN {X 0,Y 338.209,Z 468.204,A -85,B 0,C 180,E1 -14677.011,E2 -14677.011} C_VEL
LIN {X 0,Y 339.006,Z 455.932,A -85,B 0,C 180,E1 -14677.968,E2 -14677.968} C_VEL
LIN {X 0,Y 339.699,Z 443.014,A -85,B 0,C 180,E1 -14678.701,E2 -14678.701} C_VEL
LIN {X 0,Y 340.22,Z 430.381,A -85,B 0,C 180,E1 -14679.174,E2 -14679.174} C_VEL
LIN {X 0,Y 341.842,Z 352.238,A -85,B 0,C 180,E1 -14680.812,E2 -14680.812} C_VEL
LIN {X 0,Y 338.146,Z 331.141,A -85,B 0,C 180,E1 -14681.488,E2 -14681.488} C_VEL
LIN {X 0,Y 335.669,Z 323.553,A -85,B 0,C 180,E1 -14681.809,E2 -14681.809} C_VEL
LIN {X 0,Y 333.808,Z 313.906,A -85,B 0,C 180,E1 -14684.633,E2 -14684.633} C_VEL
LIN {X 0,Y 333.725,Z 313.913,A -85,B 0,C 180,E1 -14688.616,E2 -14688.616} C_VEL
LIN {X 0,Y 333.656,Z 313.92,A -85,B 0,C 180,E1 -14691.148,E2 -14691.148} C_VEL
LIN {X 0,Y 332.963,Z 314.012,A -85,B 0,C 180,E1 -14692.155,E2 -14692.155} C_VEL
LIN {X 0,Y 330.081,Z 314.367,A -85,B 0,C 180,E1 -14693.794,E2 -14693.794} C_VEL
LIN {X 0,Y 327.667,Z 314.666,A -85,B 0,C 180,E1 -14695.121,E2 -14695.121} C_VEL
LIN {X 0,Y 326.651,Z 314.797,A -85,B 0,C 180,E1 -14696.149,E2 -14696.149} C_VEL
LIN {X 0,Y 326.579,Z 314.8,A -85,B 0,C 180,E1 -14696.497,E2 -14696.497} C_VEL
LIN {X 0,Y 326.578,Z 314.802,A -85,B 0,C 180,E1 -14699.666,E2 -14699.666} C_VEL
LIN {X 0,Y 326.615,Z 314.799,A -85,B 0,C 180,E1 -14702.944,E2 -14702.944} C_VEL
LIN {X 0,Y 326.608,Z 314.797,A -85,B 0,C 180,E1 -14705.519,E2 -14705.519} C_VEL
LIN {X 0,Y 326.585,Z 314.802,A -85,B 0,C 180,E1 -14709.221,E2 -14709.221} C_VEL
LIN {X 0,Y 326.568,Z 314.808,A -85,B 0,C 180,E1 -14712.97,E2 -14712.97} C_VEL
LIN {X 0,Y 326.567,Z 314.807,A -85,B 0,C 180,E1 -14717.028,E2 -14717.028} C_VEL
LIN {X 0,Y 326.576,Z 314.804,A -85,B 0,C 180,E1 -14721.384,E2 -14721.384} C_VEL
LIN {X 0,Y 326.612,Z 314.798,A -85,B 0,C 180,E1 -14724.851,E2 -14724.851} C_VEL
LIN {X 0,Y 326.598,Z 314.803,A -85,B 0,C 180,E1 -14727.454,E2 -14727.454} C_VEL
LIN {X 0,Y 326.568,Z 314.802,A -85,B 0,C 180,E1 -14730.331,E2 -14730.331} C_VEL
LIN {X 0,Y 326.588,Z 314.801,A -85,B 0,C 180,E1 -14733.133,E2 -14733.133} C_VEL
LIN {X 0,Y 326.604,Z 314.8,A -85,B 0,C 180,E1 -14735.867,E2 -14735.867} C_VEL
LIN {X 0,Y 326.602,Z 314.798,A -85,B 0,C 180,E1 -14738.542,E2 -14738.542} C_VEL
LIN {X 0,Y 326.64,Z 314.795,A -85,B 0,C 180,E1 -14741.205,E2 -14741.205} C_VEL
LIN {X 0,Y 326.707,Z 314.784,A -85,B 0,C 180,E1 -14745.466,E2 -14745.466} C_VEL
LIN {X 0,Y 326.74,Z 314.781,A -85,B 0,C 180,E1 -14748.838,E2 -14748.838} C_VEL
LIN {X 0,Y 326.905,Z 314.761,A -85,B 0,C 180,E1 -14752.588,E2 -14752.588} C_VEL
LIN {X 0,Y 326.743,Z 314.777,A -85,B 0,C 180,E1 -14755.064,E2 -14755.064} C_VEL
LIN {X 0,Y 327.004,Z 314.747,A -85,B 0,C 180,E1 -14757.536,E2 -14757.536} C_VEL
LIN {X 0,Y 327.037,Z 314.744,A -85,B 0,C 180,E1 -14761.231,E2 -14761.231} C_VEL
LIN {X 0,Y 326.747,Z 314.78,A -85,B 0,C 180,E1 -14763.699,E2 -14763.699} C_VEL
LIN {X 0,Y 326.944,Z 314.755,A -85,B 0,C 180,E1 -14766.17,E2 -14766.17} C_VEL
LIN {X 0,Y 326.774,Z 314.777,A -85,B 0,C 180,E1 -14769.907,E2 -14769.907} C_VEL
LIN {X 0,Y 326.751,Z 314.779,A -85,B 0,C 180,E1 -14773.686,E2 -14773.686} C_VEL
LIN {X 0,Y 326.656,Z 314.792,A -85,B 0,C 180,E1 -14777.53,E2 -14777.53} C_VEL
LIN {X 0,Y 326.623,Z 314.796,A -85,B 0,C 180,E1 -14780.137,E2 -14780.137} C_VEL
LIN {X 0,Y 326.638,Z 314.793,A -85,B 0,C 180,E1 -14784.13,E2 -14784.13} C_VEL
LIN {X 0,Y 326.645,Z 314.792,A -85,B 0,C 180,E1 -14788.101,E2 -14788.101} C_VEL
LIN {X 0,Y 326.583,Z 314.804,A -85,B 0,C 180,E1 -14791.096,E2 -14791.096} C_VEL
LIN {X 0,Y 326.6,Z 314.799,A -85,B 0,C 180,E1 -14794.02,E2 -14794.02} C_VEL
LIN {X 0,Y 326.617,Z 314.8,A -85,B 0,C 180,E1 -14797.238,E2 -14797.238} C_VEL
LIN {X 0,Y 326.568,Z 314.804,A -85,B 0,C 180,E1 -14801.131,E2 -14801.131} C_VEL
LIN {X 0,Y 326.522,Z 314.809,A -85,B 0,C 180,E1 -14804.744,E2 -14804.744} C_VEL
LIN {X 0,Y 326.57,Z 314.806,A -85,B 0,C 180,E1 -14808.155,E2 -14808.155} C_VEL
LIN {X 0,Y 326.618,Z 314.798,A -85,B 0,C 180,E1 -14811.392,E2 -14811.392} C_VEL
LIN {X 0,Y 326.616,Z 314.798,A -85,B 0,C 180,E1 -14814.852,E2 -14814.852} C_VEL
LIN {X 0,Y 326.607,Z 314.8,A -85,B 0,C 180,E1 -14817.457,E2 -14817.457} C_VEL
LIN {X 0,Y 326.691,Z 314.832,A -85,B 0,C 180,E1 -14819.882,E2 -14819.882} C_VEL
LIN {X 0,Y 328.88,Z 325.923,A -85,B 0,C 180,E1 -14822.994,E2 -14822.994} C_VEL
LIN {X 0,Y 330.047,Z 332.553,A -85,B 0,C 180,E1 -14824.795,E2 -14824.795} C_VEL
LIN {X 0,Y 329.541,Z 339.283,A -85,B 0,C 180,E1 -14826.498,E2 -14826.498} C_VEL
LIN {X 0,Y 329.413,Z 340.615,A -85,B 0,C 180,E1 -14826.832,E2 -14826.832} C_VEL
LIN {X 0,Y 334.738,Z 378.015,A -85,B 0,C 180,E1 -14827.994,E2 -14827.994} C_VEL
LIN {X 0,Y 333.499,Z 448.967,A -85,B 0,C 180,E1 -14829.533,E2 -14829.533} C_VEL
LIN {X 0,Y 332.811,Z 462.256,A -85,B 0,C 180,E1 -14830.053,E2 -14830.053} C_VEL
LIN {X 0,Y 331.912,Z 474.447,A -85,B 0,C 180,E1 -14830.761,E2 -14830.761} C_VEL
LIN {X 0,Y 330.852,Z 486.747,A -85,B 0,C 180,E1 -14831.742,E2 -14831.742} C_VEL
LIN {X 0,Y 329.599,Z 498.376,A -85,B 0,C 180,E1 -14832.952,E2 -14832.952} C_VEL
LIN {X 0,Y 328.608,Z 508.229,A -85,B 0,C 180,E1 -14834.243,E2 -14834.243} C_VEL
LIN {X 0,Y 327.631,Z 517.411,A -85,B 0,C 180,E1 -14835.72,E2 -14835.72} C_VEL
LIN {X 0,Y 326.624,Z 526.656,A -85,B 0,C 180,E1 -14837.576,E2 -14837.576} C_VEL
LIN {X 0,Y 325.866,Z 534.084,A -85,B 0,C 180,E1 -14839.438,E2 -14839.438} C_VEL
LIN {X 0,Y 325.364,Z 540.035,A -85,B 0,C 180,E1 -14841.304,E2 -14841.304} C_VEL
LIN {X 0,Y 325.073,Z 544.717,A -85,B 0,C 180,E1 -14843.172,E2 -14843.172} C_VEL
LIN {X 0,Y 324.909,Z 548.27,A -85,B 0,C 180,E1 -14845.037,E2 -14845.037} C_VEL
LIN {X 0,Y 324.905,Z 550.074,A -85,B 0,C 180,E1 -14846.28,E2 -14846.28} C_VEL
LIN {X 0,Y 324.846,Z 551.426,A -85,B 0,C 180,E1 -14847.521,E2 -14847.521} C_VEL
LIN {X 0,Y 324.837,Z 552.382,A -85,B 0,C 180,E1 -14848.761,E2 -14848.761} C_VEL
LIN {X 0,Y 324.875,Z 552.948,A -85,B 0,C 180,E1 -14850.001,E2 -14850.001} C_VEL
LIN {X 0,Y 324.831,Z 553.091,A -85,B 0,C 180,E1 -14851.241,E2 -14851.241} C_VEL
LIN {X 0,Y 324.875,Z 552.172,A -85,B 0,C 180,E1 -14853.722,E2 -14853.722} C_VEL
LIN {X 0,Y 324.983,Z 550.124,A -85,B 0,C 180,E1 -14855.853,E2 -14855.853} C_VEL
LIN {X 0,Y 325.337,Z 546.693,A -85,B 0,C 180,E1 -14858.073,E2 -14858.073} C_VEL
LIN {X 0,Y 325.871,Z 542.677,A -85,B 0,C 180,E1 -14859.936,E2 -14859.936} C_VEL
LIN {X 0,Y 326.808,Z 536.527,A -85,B 0,C 180,E1 -14862.104,E2 -14862.104} C_VEL
LIN {X 0,Y 328.065,Z 529.846,A -85,B 0,C 180,E1 -14863.947,E2 -14863.947} C_VEL
LIN {X 0,Y 329.556,Z 521.581,A -85,B 0,C 180,E1 -14865.778,E2 -14865.778} C_VEL
LIN {X 0,Y 330.86,Z 513.123,A -85,B 0,C 180,E1 -14867.301,E2 -14867.301} C_VEL
LIN {X 0,Y 332.615,Z 502.693,A -85,B 0,C 180,E1 -14868.798,E2 -14868.798} C_VEL
LIN {X 0,Y 334.176,Z 492.396,A -85,B 0,C 180,E1 -14869.984,E2 -14869.984} C_VEL
LIN {X 0,Y 335.71,Z 481.124,A -85,B 0,C 180,E1 -14871.009,E2 -14871.009} C_VEL
LIN {X 0,Y 336.943,Z 469.636,A -85,B 0,C 180,E1 -14871.811,E2 -14871.811} C_VEL
LIN {X 0,Y 338.076,Z 456.46,A -85,B 0,C 180,E1 -14872.457,E2 -14872.457} C_VEL
LIN {X 0,Y 338.733,Z 443.746,A -85,B 0,C 180,E1 -14872.854,E2 -14872.854} C_VEL
LIN {X 0,Y 340.241,Z 379.544,A -85,B 0,C 180,E1 -14874.232,E2 -14874.232} C_VEL
LIN {X 0,Y 336.858,Z 360.736,A -85,B 0,C 180,E1 -14874.983,E2 -14874.983} C_VEL
LIN {X 0,Y 332.739,Z 342.121,A -85,B 0,C 180,E1 -14875.824,E2 -14875.824} C_VEL
LIN {X 0,Y 332.173,Z 339.999,A -85,B 0,C 180,E1 -14875.96,E2 -14875.96} C_VEL
LIN {X 0,Y 330.548,Z 331.103,A -85,B 0,C 180,E1 -14878.56,E2 -14878.56} C_VEL
LIN {X 0,Y 328.185,Z 321.106,A -85,B 0,C 180,E1 -14881.666,E2 -14881.666} C_VEL
LIN {X 0,Y 326.615,Z 314.808,A -85,B 0,C 180,E1 -14883.731,E2 -14883.731} C_VEL
LIN {X 0,Y 326.625,Z 314.8,A -85,B 0,C 180,E1 -14887.238,E2 -14887.238} C_VEL
LIN {X 0,Y 326.576,Z 314.803,A -85,B 0,C 180,E1 -14891.131,E2 -14891.131} C_VEL
LIN {X 0,Y 326.529,Z 314.813,A -85,B 0,C 180,E1 -14894.743,E2 -14894.743} C_VEL
LIN {X 0,Y 326.576,Z 314.805,A -85,B 0,C 180,E1 -14898.154,E2 -14898.154} C_VEL
LIN {X 0,Y 326.588,Z 314.797,A -85,B 0,C 180,E1 -14901.386,E2 -14901.386} C_VEL
LIN {X 0,Y 326.621,Z 314.795,A -85,B 0,C 180,E1 -14904.852,E2 -14904.852} C_VEL
LIN {X 0,Y 326.609,Z 314.795,A -85,B 0,C 180,E1 -14907.456,E2 -14907.456} C_VEL
LIN {X 0,Y 326.626,Z 314.798,A -85,B 0,C 180,E1 -14910.338,E2 -14910.338} C_VEL
LIN {X 0,Y 326.63,Z 314.801,A -85,B 0,C 180,E1 -14913.138,E2 -14913.138} C_VEL
LIN {X 0,Y 326.644,Z 314.793,A -85,B 0,C 180,E1 -14915.871,E2 -14915.871} C_VEL
LIN {X 0,Y 326.625,Z 314.796,A -85,B 0,C 180,E1 -14919.863,E2 -14919.863} C_VEL
LIN {X 0,Y 326.72,Z 314.781,A -85,B 0,C 180,E1 -14923.761,E2 -14923.761} C_VEL
LIN {X 0,Y 326.761,Z 314.775,A -85,B 0,C 180,E1 -14926.315,E2 -14926.315} C_VEL
LIN {X 0,Y 326.806,Z 314.771,A -85,B 0,C 180,E1 -14930.094,E2 -14930.094} C_VEL
LIN {X 0,Y 326.982,Z 314.753,A -85,B 0,C 180,E1 -14933.831,E2 -14933.831} C_VEL
LIN {X 0,Y 327.018,Z 314.743,A -85,B 0,C 180,E1 -14937.537,E2 -14937.537} C_VEL
LIN {X 0,Y 327.143,Z 314.725,A -85,B 0,C 180,E1 -14940,E2 -14940} C_VEL
LIN {X 0,Y 327.037,Z 314.746,A -85,B 0,C 180,E1 -14942.464,E2 -14942.464} C_VEL
LIN {X 0,Y 326.931,Z 314.754,A -85,B 0,C 180,E1 -14946.502,E2 -14946.502} C_VEL
LIN {X 0,Y 326.785,Z 314.771,A -85,B 0,C 180,E1 -14949.907,E2 -14949.907} C_VEL
LIN {X 0,Y 326.762,Z 314.773,A -85,B 0,C 180,E1 -14953.686,E2 -14953.686} C_VEL
LIN {X 0,Y 326.666,Z 314.785,A -85,B 0,C 180,E1 -14957.53,E2 -14957.53} C_VEL
LIN {X 0,Y 326.636,Z 314.795,A -85,B 0,C 180,E1 -14960.137,E2 -14960.137} C_VEL
LIN {X 0,Y 326.646,Z 314.792,A -85,B 0,C 180,E1 -14964.13,E2 -14964.13} C_VEL
LIN {X 0,Y 326.631,Z 314.791,A -85,B 0,C 180,E1 -14968.253,E2 -14968.253} C_VEL
LIN {X 0,Y 326.578,Z 314.802,A -85,B 0,C 180,E1 -14971.097,E2 -14971.097} C_VEL
LIN {X 0,Y 326.61,Z 314.796,A -85,B 0,C 180,E1 -14974.02,E2 -14974.02} C_VEL
LIN {X 0,Y 326.63,Z 314.796,A -85,B 0,C 180,E1 -14977.238,E2 -14977.238} C_VEL
LIN {X 0,Y 326.58,Z 314.806,A -85,B 0,C 180,E1 -14981.131,E2 -14981.131} C_VEL
LIN {X 0,Y 326.53,Z 314.812,A -85,B 0,C 180,E1 -14984.743,E2 -14984.743} C_VEL
LIN {X 0,Y 326.566,Z 314.81,A -85,B 0,C 180,E1 -14988.152,E2 -14988.152} C_VEL
LIN {X 0,Y 326.59,Z 314.911,A -85,B 0,C 180,E1 -14989.746,E2 -14989.746} C_VEL
LIN {X 0,Y 328.869,Z 324.111,A -85,B 0,C 180,E1 -14992.775,E2 -14992.775} C_VEL
LIN {X 0,Y 337.887,Z 344.08,A -85,B 0,C 180,E1 -14994.142,E2 -14994.142} C_VEL
LIN {X 0,Y 339.151,Z 347.924,A -85,B 0,C 180,E1 -14994.351,E2 -14994.351} C_VEL
LIN {X 0,Y 340.83,Z 355.564,A -85,B 0,C 180,E1 -14994.685,E2 -14994.685} C_VEL
LIN {X 0,Y 338.805,Z 432.239,A -85,B 0,C 180,E1 -14996.348,E2 -14996.348} C_VEL
LIN {X 0,Y 338.063,Z 444.723,A -85,B 0,C 180,E1 -14996.84,E2 -14996.84} C_VEL
LIN {X 0,Y 336.899,Z 457.74,A -85,B 0,C 180,E1 -14997.597,E2 -14997.597} C_VEL
LIN {X 0,Y 335.817,Z 468.437,A -85,B 0,C 180,E1 -14998.452,E2 -14998.452} C_VEL
LIN {X 0,Y 334.299,Z 480.467,A -85,B 0,C 180,E1 -14999.698,E2 -14999.698} C_VEL
LIN {X 0,Y 332.619,Z 491.187,A -85,B 0,C 180,E1 -15001.096,E2 -15001.096} C_VEL
LIN {X 0,Y 331.082,Z 500.057,A -85,B 0,C 180,E1 -15002.537,E2 -15002.537} C_VEL
LIN {X 0,Y 329.737,Z 507.835,A -85,B 0,C 180,E1 -15004.091,E2 -15004.091} C_VEL
LIN {X 0,Y 328.243,Z 515.544,A -85,B 0,C 180,E1 -15005.995,E2 -15005.995} C_VEL
LIN {X 0,Y 327.165,Z 521.767,A -85,B 0,C 180,E1 -15007.944,E2 -15007.944} C_VEL
LIN {X 0,Y 326.265,Z 526.508,A -85,B 0,C 180,E1 -15009.839,E2 -15009.839} C_VEL
LIN {X 0,Y 325.688,Z 530.055,A -85,B 0,C 180,E1 -15011.71,E2 -15011.71} C_VEL
LIN {X 0,Y 325.157,Z 532.716,A -85,B 0,C 180,E1 -15013.68,E2 -15013.68} C_VEL
LIN {X 0,Y 324.981,Z 533.895,A -85,B 0,C 180,E1 -15014.958,E2 -15014.958} C_VEL
LIN {X 0,Y 324.882,Z 534.814,A -85,B 0,C 180,E1 -15016.773,E2 -15016.773} C_VEL
LIN {X 0,Y 324.748,Z 534.868,A -85,B 0,C 180,E1 -15018.768,E2 -15018.768} C_VEL
LIN {X 0,Y 324.686,Z 534.383,A -85,B 0,C 180,E1 -15020.027,E2 -15020.027} C_VEL
LIN {X 0,Y 324.765,Z 533.466,A -85,B 0,C 180,E1 -15021.286,E2 -15021.286} C_VEL
LIN {X 0,Y 324.874,Z 532.154,A -85,B 0,C 180,E1 -15022.541,E2 -15022.541} C_VEL
LIN {X 0,Y 325.049,Z 530.034,A -85,B 0,C 180,E1 -15024.038,E2 -15024.038} C_VEL
LIN {X 0,Y 325.347,Z 525.602,A -85,B 0,C 180,E1 -15026.284,E2 -15026.284} C_VEL
LIN {X 0,Y 325.803,Z 520.695,A -85,B 0,C 180,E1 -15028.145,E2 -15028.145} C_VEL
LIN {X 0,Y 326.358,Z 514.534,A -85,B 0,C 180,E1 -15029.999,E2 -15029.999} C_VEL
LIN {X 0,Y 327.344,Z 506.836,A -85,B 0,C 180,E1 -15031.845,E2 -15031.845} C_VEL
LIN {X 0,Y 328.276,Z 497.223,A -85,B 0,C 180,E1 -15033.682,E2 -15033.682} C_VEL
LIN {X 0,Y 329.384,Z 488.329,A -85,B 0,C 180,E1 -15035.048,E2 -15035.048} C_VEL
LIN {X 0,Y 330.601,Z 477.409,A -85,B 0,C 180,E1 -15036.407,E2 -15036.407} C_VEL
LIN {X 0,Y 331.606,Z 465.007,A -85,B 0,C 180,E1 -15037.611,E2 -15037.611} C_VEL
LIN {X 0,Y 332.38,Z 452.852,A -85,B 0,C 180,E1 -15038.511,E2 -15038.511} C_VEL
LIN {X 0,Y 333.048,Z 440.014,A -85,B 0,C 180,E1 -15039.182,E2 -15039.182} C_VEL
LIN {X 0,Y 333.604,Z 426.312,A -85,B 0,C 180,E1 -15039.625,E2 -15039.625} C_VEL
LIN {X 0,Y 335.053,Z 352.751,A -85,B 0,C 180,E1 -15041.187,E2 -15041.187} C_VEL
LIN {X 0,Y 331.608,Z 333.101,A -85,B 0,C 180,E1 -15041.833,E2 -15041.833} C_VEL
LIN {X 0,Y 328.521,Z 323.715,A -85,B 0,C 180,E1 -15042.253,E2 -15042.253} C_VEL
LIN {X 0,Y 326.739,Z 314.786,A -85,B 0,C 180,E1 -15044.886,E2 -15044.886} C_VEL
LIN {X 0,Y 326.663,Z 314.793,A -85,B 0,C 180,E1 -15048.826,E2 -15048.826} C_VEL
LIN {X 0,Y 326.593,Z 314.801,A -85,B 0,C 180,E1 -15052.788,E2 -15052.788} C_VEL
LIN {X 0,Y 326.579,Z 314.8,A -85,B 0,C 180,E1 -15056.497,E2 -15056.497} C_VEL
LIN {X 0,Y 325.94,Z 314.885,A -85,B 0,C 180,E1 -15057.525,E2 -15057.525} C_VEL
LIN {X 0,Y 323.095,Z 315.245,A -85,B 0,C 180,E1 -15059.199,E2 -15059.199} C_VEL
LIN {X 0,Y 320.661,Z 315.547,A -85,B 0,C 180,E1 -15060.555,E2 -15060.555} C_VEL
LIN {X 0,Y 319.608,Z 315.672,A -85,B 0,C 180,E1 -15061.606,E2 -15061.606} C_VEL
LIN {X 0,Y 319.518,Z 315.681,A -85,B 0,C 180,E1 -15061.962,E2 -15061.962} C_VEL
LIN {X 0,Y 319.576,Z 315.673,A -85,B 0,C 180,E1 -15065.541,E2 -15065.541} C_VEL
LIN {X 0,Y 319.525,Z 315.679,A -85,B 0,C 180,E1 -15069.661,E2 -15069.661} C_VEL
LIN {X 0,Y 319.514,Z 315.682,A -85,B 0,C 180,E1 -15073.459,E2 -15073.459} C_VEL
LIN {X 0,Y 319.545,Z 315.68,A -85,B 0,C 180,E1 -15077.014,E2 -15077.014} C_VEL
LIN {X 0,Y 319.54,Z 315.678,A -85,B 0,C 180,E1 -15080.369,E2 -15080.369} C_VEL
LIN {X 0,Y 319.572,Z 315.672,A -85,B 0,C 180,E1 -15084.457,E2 -15084.457} C_VEL
LIN {X 0,Y 319.513,Z 315.681,A -85,B 0,C 180,E1 -15088.136,E2 -15088.136} C_VEL
LIN {X 0,Y 319.535,Z 315.681,A -85,B 0,C 180,E1 -15091.613,E2 -15091.613} C_VEL
LIN {X 0,Y 319.534,Z 315.679,A -85,B 0,C 180,E1 -15095.298,E2 -15095.298} C_VEL
LIN {X 0,Y 319.556,Z 315.678,A -85,B 0,C 180,E1 -15098.044,E2 -15098.044} C_VEL
LIN {X 0,Y 319.575,Z 315.675,A -85,B 0,C 180,E1 -15102.068,E2 -15102.068} C_VEL
LIN {X 0,Y 319.685,Z 315.663,A -85,B 0,C 180,E1 -15106.005,E2 -15106.005} C_VEL
LIN {X 0,Y 319.723,Z 315.66,A -85,B 0,C 180,E1 -15109.871,E2 -15109.871} C_VEL
LIN {X 0,Y 319.89,Z 315.635,A -85,B 0,C 180,E1 -15113.693,E2 -15113.693} C_VEL
LIN {X 0,Y 319.951,Z 315.625,A -85,B 0,C 180,E1 -15117.482,E2 -15117.482} C_VEL
LIN {X 0,Y 320.004,Z 315.62,A -85,B 0,C 180,E1 -15121.258,E2 -15121.258} C_VEL
LIN {X 0,Y 319.715,Z 315.654,A -85,B 0,C 180,E1 -15125.044,E2 -15125.044} C_VEL
LIN {X 0,Y 319.872,Z 315.635,A -85,B 0,C 180,E1 -15127.575,E2 -15127.575} C_VEL
LIN {X 0,Y 319.706,Z 315.658,A -85,B 0,C 180,E1 -15131.411,E2 -15131.411} C_VEL
LIN {X 0,Y 319.704,Z 315.661,A -85,B 0,C 180,E1 -15134.711,E2 -15134.711} C_VEL
LIN {X 0,Y 319.632,Z 315.672,A -85,B 0,C 180,E1 -15139.012,E2 -15139.012} C_VEL
LIN {X 0,Y 319.551,Z 315.68,A -85,B 0,C 180,E1 -15143.321,E2 -15143.321} C_VEL
LIN {X 0,Y 319.587,Z 315.672,A -85,B 0,C 180,E1 -15146.092,E2 -15146.092} C_VEL
LIN {X 0,Y 319.571,Z 315.676,A -85,B 0,C 180,E1 -15148.935,E2 -15148.935} C_VEL
LIN {X 0,Y 319.524,Z 315.681,A -85,B 0,C 180,E1 -15151.863,E2 -15151.863} C_VEL
LIN {X 0,Y 319.573,Z 315.679,A -85,B 0,C 180,E1 -15155.544,E2 -15155.544} C_VEL
LIN {X 0,Y 319.553,Z 315.681,A -85,B 0,C 180,E1 -15159.67,E2 -15159.67} C_VEL
LIN {X 0,Y 319.515,Z 315.683,A -85,B 0,C 180,E1 -15163.461,E2 -15163.461} C_VEL
LIN {X 0,Y 319.548,Z 315.678,A -85,B 0,C 180,E1 -15167.017,E2 -15167.017} C_VEL
LIN {X 0,Y 319.542,Z 315.68,A -85,B 0,C 180,E1 -15170.372,E2 -15170.372} C_VEL
LIN {X 0,Y 319.554,Z 315.679,A -85,B 0,C 180,E1 -15173.573,E2 -15173.573} C_VEL
LIN {X 0,Y 319.574,Z 315.677,A -85,B 0,C 180,E1 -15176.687,E2 -15176.687} C_VEL
LIN {X 0,Y 319.635,Z 315.698,A -85,B 0,C 180,E1 -15179.553,E2 -15179.553} C_VEL
LIN {X 0,Y 321.83,Z 326.65,A -85,B 0,C 180,E1 -15182.705,E2 -15182.705} C_VEL
LIN {X 0,Y 323.123,Z 334.599,A -85,B 0,C 180,E1 -15184.906,E2 -15184.906} C_VEL
LIN {X 0,Y 322.56,Z 340.407,A -85,B 0,C 180,E1 -15186.399,E2 -15186.399} C_VEL
LIN {X 0,Y 328.017,Z 379.575,A -85,B 0,C 180,E1 -15187.644,E2 -15187.644} C_VEL
LIN {X 0,Y 326.72,Z 448.701,A -85,B 0,C 180,E1 -15189.171,E2 -15189.171} C_VEL
LIN {X 0,Y 326.005,Z 462.011,A -85,B 0,C 180,E1 -15189.7,E2 -15189.7} C_VEL
LIN {X 0,Y 325.08,Z 474.214,A -85,B 0,C 180,E1 -15190.423,E2 -15190.423} C_VEL
LIN {X 0,Y 324.098,Z 485.72,A -85,B 0,C 180,E1 -15191.347,E2 -15191.347} C_VEL
LIN {X 0,Y 322.793,Z 497.509,A -85,B 0,C 180,E1 -15192.581,E2 -15192.581} C_VEL
LIN {X 0,Y 321.637,Z 508.427,A -85,B 0,C 180,E1 -15194.036,E2 -15194.036} C_VEL
LIN {X 0,Y 320.733,Z 516.758,A -85,B 0,C 180,E1 -15195.406,E2 -15195.406} C_VEL
LIN {X 0,Y 319.791,Z 524.716,A -85,B 0,C 180,E1 -15196.983,E2 -15196.983} C_VEL
LIN {X 0,Y 318.92,Z 532.471,A -85,B 0,C 180,E1 -15198.884,E2 -15198.884} C_VEL
LIN {X 0,Y 318.322,Z 539.609,A -85,B 0,C 180,E1 -15201.11,E2 -15201.11} C_VEL
LIN {X 0,Y 317.998,Z 544.341,A -85,B 0,C 180,E1 -15203.019,E2 -15203.019} C_VEL
LIN {X 0,Y 317.82,Z 547.94,A -85,B 0,C 180,E1 -15204.926,E2 -15204.926} C_VEL
LIN {X 0,Y 317.813,Z 549.784,A -85,B 0,C 180,E1 -15206.197,E2 -15206.197} C_VEL
LIN {X 0,Y 317.767,Z 551.159,A -85,B 0,C 180,E1 -15207.466,E2 -15207.466} C_VEL
LIN {X 0,Y 317.748,Z 552.134,A -85,B 0,C 180,E1 -15208.734,E2 -15208.734} C_VEL
LIN {X 0,Y 317.783,Z 552.719,A -85,B 0,C 180,E1 -15210.001,E2 -15210.001} C_VEL
LIN {X 0,Y 317.742,Z 552.9,A -85,B 0,C 180,E1 -15211.268,E2 -15211.268} C_VEL
LIN {X 0,Y 317.754,Z 552.654,A -85,B 0,C 180,E1 -15212.536,E2 -15212.536} C_VEL
LIN {X 0,Y 317.786,Z 552.022,A -85,B 0,C 180,E1 -15213.805,E2 -15213.805} C_VEL
LIN {X 0,Y 317.881,Z 550.243,A -85,B 0,C 180,E1 -15215.788,E2 -15215.788} C_VEL
LIN {X 0,Y 318.278,Z 546.638,A -85,B 0,C 180,E1 -15218.253,E2 -15218.253} C_VEL
LIN {X 0,Y 318.866,Z 542.665,A -85,B 0,C 180,E1 -15220.157,E2 -15220.157} C_VEL
LIN {X 0,Y 319.708,Z 537.576,A -85,B 0,C 180,E1 -15222.055,E2 -15222.055} C_VEL
LIN {X 0,Y 320.91,Z 531.191,A -85,B 0,C 180,E1 -15223.941,E2 -15223.941} C_VEL
LIN {X 0,Y 322.464,Z 523.242,A -85,B 0,C 180,E1 -15225.81,E2 -15225.81} C_VEL
LIN {X 0,Y 323.838,Z 514.913,A -85,B 0,C 180,E1 -15227.41,E2 -15227.41} C_VEL
LIN {X 0,Y 325.518,Z 505.344,A -85,B 0,C 180,E1 -15228.897,E2 -15228.897} C_VEL
LIN {X 0,Y 327.332,Z 494.34,A -85,B 0,C 180,E1 -15230.257,E2 -15230.257} C_VEL
LIN {X 0,Y 328.89,Z 483.581,A -85,B 0,C 180,E1 -15231.302,E2 -15231.302} C_VEL
LIN {X 0,Y 330.262,Z 471.755,A -85,B 0,C 180,E1 -15232.193,E2 -15232.193} C_VEL
LIN {X 0,Y 331.553,Z 458.984,A -85,B 0,C 180,E1 -15232.883,E2 -15232.883} C_VEL
LIN {X 0,Y 332.276,Z 446.601,A -85,B 0,C 180,E1 -15233.324,E2 -15233.324} C_VEL
LIN {X 0,Y 333.993,Z 380.866,A -85,B 0,C 180,E1 -15234.766,E2 -15234.766} C_VEL
LIN {X 0,Y 330.769,Z 362.695,A -85,B 0,C 180,E1 -15235.512,E2 -15235.512} C_VEL
LIN {X 0,Y 326.791,Z 344.55,A -85,B 0,C 180,E1 -15236.354,E2 -15236.354} C_VEL
LIN {X 0,Y 324.993,Z 339.778,A -85,B 0,C 180,E1 -15236.683,E2 -15236.683} C_VEL
LIN {X 0,Y 323.617,Z 332.442,A -85,B 0,C 180,E1 -15238.893,E2 -15238.893} C_VEL
LIN {X 0,Y 321.301,Z 322.587,A -85,B 0,C 180,E1 -15242.036,E2 -15242.036} C_VEL
LIN {X 0,Y 319.563,Z 315.683,A -85,B 0,C 180,E1 -15244.398,E2 -15244.398} C_VEL
LIN {X 0,Y 319.537,Z 315.682,A -85,B 0,C 180,E1 -15248.014,E2 -15248.014} C_VEL
LIN {X 0,Y 319.525,Z 315.681,A -85,B 0,C 180,E1 -15251.597,E2 -15251.597} C_VEL
LIN {X 0,Y 319.49,Z 315.687,A -85,B 0,C 180,E1 -15255.257,E2 -15255.257} C_VEL
LIN {X 0,Y 319.527,Z 315.68,A -85,B 0,C 180,E1 -15258.712,E2 -15258.712} C_VEL
LIN {X 0,Y 319.549,Z 315.676,A -85,B 0,C 180,E1 -15262.352,E2 -15262.352} C_VEL
LIN {X 0,Y 319.561,Z 315.675,A -85,B 0,C 180,E1 -15265.124,E2 -15265.124} C_VEL
LIN {X 0,Y 319.526,Z 315.676,A -85,B 0,C 180,E1 -15268.138,E2 -15268.138} C_VEL
LIN {X 0,Y 319.595,Z 315.669,A -85,B 0,C 180,E1 -15271.597,E2 -15271.597} C_VEL
LIN {X 0,Y 319.584,Z 315.671,A -85,B 0,C 180,E1 -15275.302,E2 -15275.302} C_VEL
LIN {X 0,Y 319.569,Z 315.674,A -85,B 0,C 180,E1 -15278.046,E2 -15278.046} C_VEL
LIN {X 0,Y 319.616,Z 315.667,A -85,B 0,C 180,E1 -15282.071,E2 -15282.071} C_VEL
LIN {X 0,Y 319.734,Z 315.652,A -85,B 0,C 180,E1 -15286.008,E2 -15286.008} C_VEL
LIN {X 0,Y 319.753,Z 315.652,A -85,B 0,C 180,E1 -15289.873,E2 -15289.873} C_VEL
LIN {X 0,Y 319.936,Z 315.628,A -85,B 0,C 180,E1 -15293.694,E2 -15293.694} C_VEL
LIN {X 0,Y 320.017,Z 315.616,A -85,B 0,C 180,E1 -15298.742,E2 -15298.742} C_VEL
LIN {X 0,Y 320.018,Z 315.612,A -85,B 0,C 180,E1 -15301.259,E2 -15301.259} C_VEL
LIN {X 0,Y 319.722,Z 315.655,A -85,B 0,C 180,E1 -15303.781,E2 -15303.781} C_VEL
LIN {X 0,Y 319.896,Z 315.632,A -85,B 0,C 180,E1 -15306.487,E2 -15306.487} C_VEL
LIN {X 0,Y 319.738,Z 315.65,A -85,B 0,C 180,E1 -15310.128,E2 -15310.128} C_VEL
LIN {X 0,Y 319.735,Z 315.649,A -85,B 0,C 180,E1 -15313.992,E2 -15313.992} C_VEL
LIN {X 0,Y 319.627,Z 315.661,A -85,B 0,C 180,E1 -15317.929,E2 -15317.929} C_VEL
LIN {X 0,Y 319.591,Z 315.672,A -85,B 0,C 180,E1 -15320.601,E2 -15320.601} C_VEL
LIN {X 0,Y 319.561,Z 315.677,A -85,B 0,C 180,E1 -15323.321,E2 -15323.321} C_VEL
LIN {X 0,Y 319.582,Z 315.671,A -85,B 0,C 180,E1 -15326.093,E2 -15326.093} C_VEL
LIN {X 0,Y 319.561,Z 315.672,A -85,B 0,C 180,E1 -15328.937,E2 -15328.937} C_VEL
LIN {X 0,Y 319.528,Z 315.678,A -85,B 0,C 180,E1 -15331.863,E2 -15331.863} C_VEL
LIN {X 0,Y 319.583,Z 315.676,A -85,B 0,C 180,E1 -15335.543,E2 -15335.543} C_VEL
LIN {X 0,Y 319.56,Z 315.679,A -85,B 0,C 180,E1 -15338.01,E2 -15338.01} C_VEL
LIN {X 0,Y 319.528,Z 315.682,A -85,B 0,C 180,E1 -15341.597,E2 -15341.597} C_VEL
LIN {X 0,Y 319.491,Z 315.69,A -85,B 0,C 180,E1 -15345.257,E2 -15345.257} C_VEL
LIN {X 0,Y 319.508,Z 315.69,A -85,B 0,C 180,E1 -15348.407,E2 -15348.407} C_VEL
LIN {X 0,Y 319.535,Z 315.751,A -85,B 0,C 180,E1 -15349.106,E2 -15349.106} C_VEL
LIN {X 0,Y 321.768,Z 324.524,A -85,B 0,C 180,E1 -15352.043,E2 -15352.043} C_VEL
LIN {X 0,Y 330.904,Z 344.182,A -85,B 0,C 180,E1 -15353.475,E2 -15353.475} C_VEL
LIN {X 0,Y 333.053,Z 349.732,A -85,B 0,C 180,E1 -15353.819,E2 -15353.819} C_VEL
LIN {X 0,Y 334.581,Z 357.506,A -85,B 0,C 180,E1 -15354.154,E2 -15354.154} C_VEL
LIN {X 0,Y 332.512,Z 432.065,A -85,B 0,C 180,E1 -15355.795,E2 -15355.795} C_VEL
LIN {X 0,Y 331.748,Z 444.051,A -85,B 0,C 180,E1 -15356.261,E2 -15356.261} C_VEL
LIN {X 0,Y 330.623,Z 456.723,A -85,B 0,C 180,E1 -15356.995,E2 -15356.995} C_VEL
LIN {X 0,Y 329.323,Z 468.753,A -85,B 0,C 180,E1 -15357.954,E2 -15357.954} C_VEL
LIN {X 0,Y 327.835,Z 480.234,A -85,B 0,C 180,E1 -15359.162,E2 -15359.162} C_VEL
LIN {X 0,Y 326.023,Z 491.351,A -85,B 0,C 180,E1 -15360.631,E2 -15360.631} C_VEL
LIN {X 0,Y 324.271,Z 500.902,A -85,B 0,C 180,E1 -15362.226,E2 -15362.226} C_VEL
LIN {X 0,Y 322.562,Z 510.097,A -85,B 0,C 180,E1 -15364.166,E2 -15364.166} C_VEL
LIN {X 0,Y 321.134,Z 517.43,A -85,B 0,C 180,E1 -15366.116,E2 -15366.116} C_VEL
LIN {X 0,Y 320.011,Z 523.206,A -85,B 0,C 180,E1 -15368.077,E2 -15368.077} C_VEL
LIN {X 0,Y 319.128,Z 527.707,A -85,B 0,C 180,E1 -15370.04,E2 -15370.04} C_VEL
LIN {X 0,Y 318.517,Z 531.072,A -85,B 0,C 180,E1 -15372.006,E2 -15372.006} C_VEL
LIN {X 0,Y 318.161,Z 532.727,A -85,B 0,C 180,E1 -15373.311,E2 -15373.311} C_VEL
LIN {X 0,Y 317.921,Z 533.964,A -85,B 0,C 180,E1 -15374.616,E2 -15374.616} C_VEL
LIN {X 0,Y 317.812,Z 535.02,A -85,B 0,C 180,E1 -15376.659,E2 -15376.659} C_VEL
LIN {X 0,Y 317.681,Z 535.09,A -85,B 0,C 180,E1 -15378.515,E2 -15378.515} C_VEL
LIN {X 0,Y 317.589,Z 534.674,A -85,B 0,C 180,E1 -15379.802,E2 -15379.802} C_VEL
LIN {X 0,Y 317.672,Z 533.812,A -85,B 0,C 180,E1 -15381.09,E2 -15381.09} C_VEL
LIN {X 0,Y 317.758,Z 532.544,A -85,B 0,C 180,E1 -15382.373,E2 -15382.373} C_VEL
LIN {X 0,Y 317.961,Z 530.22,A -85,B 0,C 180,E1 -15384.077,E2 -15384.077} C_VEL
LIN {X 0,Y 318.254,Z 526.168,A -85,B 0,C 180,E1 -15386.201,E2 -15386.201} C_VEL
LIN {X 0,Y 318.704,Z 521.359,A -85,B 0,C 180,E1 -15388.104,E2 -15388.104} C_VEL
LIN {X 0,Y 319.249,Z 515.307,A -85,B 0,C 180,E1 -15389.999,E2 -15389.999} C_VEL
LIN {X 0,Y 320.271,Z 507.758,A -85,B 0,C 180,E1 -15391.885,E2 -15391.885} C_VEL
LIN {X 0,Y 321.076,Z 500.078,A -85,B 0,C 180,E1 -15393.45,E2 -15393.45} C_VEL
LIN {X 0,Y 322.112,Z 490.706,A -85,B 0,C 180,E1 -15395.006,E2 -15395.006} C_VEL
LIN {X 0,Y 323.43,Z 480.257,A -85,B 0,C 180,E1 -15396.393,E2 -15396.393} C_VEL
LIN {X 0,Y 324.492,Z 468.703,A -85,B 0,C 180,E1 -15397.622,E2 -15397.622} C_VEL
LIN {X 0,Y 325.353,Z 456.469,A -85,B 0,C 180,E1 -15398.618,E2 -15398.618} C_VEL
LIN {X 0,Y 326.094,Z 443.597,A -85,B 0,C 180,E1 -15399.379,E2 -15399.379} C_VEL
LIN {X 0,Y 326.65,Z 431.082,A -85,B 0,C 180,E1 -15399.871,E2 -15399.871} C_VEL
LIN {X 0,Y 328.333,Z 353.617,A -85,B 0,C 180,E1 -15401.565,E2 -15401.565} C_VEL
LIN {X 0,Y 325.154,Z 335.338,A -85,B 0,C 180,E1 -15402.181,E2 -15402.181} C_VEL
LIN {X 0,Y 321.34,Z 323.895,A -85,B 0,C 180,E1 -15402.712,E2 -15402.712} C_VEL
LIN {X 0,Y 319.68,Z 315.665,A -85,B 0,C 180,E1 -15405.208,E2 -15405.208} C_VEL
LIN {X 0,Y 319.589,Z 315.674,A -85,B 0,C 180,E1 -15409.259,E2 -15409.259} C_VEL
LIN {X 0,Y 319.543,Z 315.678,A -85,B 0,C 180,E1 -15413.32,E2 -15413.32} C_VEL
LIN {X 0,Y 319.526,Z 315.681,A -85,B 0,C 180,E1 -15416.487,E2 -15416.487} C_VEL
LIN {X 0,Y 319.551,Z 315.682,A -85,B 0,C 180,E1 -15420.386,E2 -15420.386} C_VEL
LIN {X 0,Y 319.518,Z 315.681,A -85,B 0,C 180,E1 -15421.962,E2 -15421.962} C_VEL
LIN {X 0,Y 318.854,Z 315.765,A -85,B 0,C 180,E1 -15423.014,E2 -15423.014} C_VEL
LIN {X 0,Y 316.045,Z 316.118,A -85,B 0,C 180,E1 -15424.727,E2 -15424.727} C_VEL
LIN {X 0,Y 313.651,Z 316.415,A -85,B 0,C 180,E1 -15426.116,E2 -15426.116} C_VEL
LIN {X 0,Y 312.599,Z 316.545,A -85,B 0,C 180,E1 -15427.19,E2 -15427.19} C_VEL
LIN {X 0,Y 312.499,Z 316.556,A -85,B 0,C 180,E1 -15427.554,E2 -15427.554} C_VEL
LIN {X 0,Y 312.437,Z 316.566,A -85,B 0,C 180,E1 -15430.716,E2 -15430.716} C_VEL
LIN {X 0,Y 312.446,Z 316.563,A -85,B 0,C 180,E1 -15434.209,E2 -15434.209} C_VEL
LIN {X 0,Y 312.449,Z 316.559,A -85,B 0,C 180,E1 -15437.924,E2 -15437.924} C_VEL
LIN {X 0,Y 312.478,Z 316.557,A -85,B 0,C 180,E1 -15441.922,E2 -15441.922} C_VEL
LIN {X 0,Y 312.524,Z 316.549,A -85,B 0,C 180,E1 -15444.219,E2 -15444.219} C_VEL
LIN {X 0,Y 312.493,Z 316.56,A -85,B 0,C 180,E1 -15447.332,E2 -15447.332} C_VEL
LIN {X 0,Y 312.475,Z 316.563,A -85,B 0,C 180,E1 -15451.299,E2 -15451.299} C_VEL
LIN {X 0,Y 312.514,Z 316.549,A -85,B 0,C 180,E1 -15454.704,E2 -15454.704} C_VEL
LIN {X 0,Y 312.533,Z 316.555,A -85,B 0,C 180,E1 -15457.524,E2 -15457.524} C_VEL
LIN {X 0,Y 312.541,Z 316.555,A -85,B 0,C 180,E1 -15461.65,E2 -15461.65} C_VEL
LIN {X 0,Y 312.629,Z 316.538,A -85,B 0,C 180,E1 -15465.683,E2 -15465.683} C_VEL
LIN {X 0,Y 312.673,Z 316.536,A -85,B 0,C 180,E1 -15469.641,E2 -15469.641} C_VEL
LIN {X 0,Y 312.832,Z 316.513,A -85,B 0,C 180,E1 -15473.55,E2 -15473.55} C_VEL
LIN {X 0,Y 312.899,Z 316.503,A -85,B 0,C 180,E1 -15477.425,E2 -15477.425} C_VEL
LIN {X 0,Y 312.971,Z 316.496,A -85,B 0,C 180,E1 -15481.286,E2 -15481.286} C_VEL
LIN {X 0,Y 312.844,Z 316.512,A -85,B 0,C 180,E1 -15486.449,E2 -15486.449} C_VEL
LIN {X 0,Y 312.742,Z 316.527,A -85,B 0,C 180,E1 -15489.05,E2 -15489.05} C_VEL
LIN {X 0,Y 312.626,Z 316.541,A -85,B 0,C 180,E1 -15492.991,E2 -15492.991} C_VEL
LIN {X 0,Y 312.613,Z 316.537,A -85,B 0,C 180,E1 -15495.651,E2 -15495.651} C_VEL
LIN {X 0,Y 312.552,Z 316.549,A -85,B 0,C 180,E1 -15499.712,E2 -15499.712} C_VEL
LIN {X 0,Y 312.518,Z 316.556,A -85,B 0,C 180,E1 -15502.781,E2 -15502.781} C_VEL
LIN {X 0,Y 312.564,Z 316.547,A -85,B 0,C 180,E1 -15505.924,E2 -15505.924} C_VEL
LIN {X 0,Y 312.53,Z 316.554,A -85,B 0,C 180,E1 -15509.651,E2 -15509.651} C_VEL
LIN {X 0,Y 312.513,Z 316.557,A -85,B 0,C 180,E1 -15513.69,E2 -15513.69} C_VEL
LIN {X 0,Y 312.509,Z 316.558,A -85,B 0,C 180,E1 -15517.387,E2 -15517.387} C_VEL
LIN {X 0,Y 312.482,Z 316.557,A -85,B 0,C 180,E1 -15520.71,E2 -15520.71} C_VEL
LIN {X 0,Y 312.446,Z 316.564,A -85,B 0,C 180,E1 -15524.211,E2 -15524.211} C_VEL
LIN {X 0,Y 312.478,Z 316.563,A -85,B 0,C 180,E1 -15527.92,E2 -15527.92} C_VEL
LIN {X 0,Y 312.53,Z 316.557,A -85,B 0,C 180,E1 -15531.912,E2 -15531.912} C_VEL
LIN {X 0,Y 312.503,Z 316.559,A -85,B 0,C 180,E1 -15535.791,E2 -15535.791} C_VEL
LIN {X 0,Y 312.574,Z 316.66,A -85,B 0,C 180,E1 -15539.236,E2 -15539.236} C_VEL
LIN {X 0,Y 314.935,Z 328.283,A -85,B 0,C 180,E1 -15542.663,E2 -15542.663} C_VEL
LIN {X 0,Y 316.13,Z 335.335,A -85,B 0,C 180,E1 -15544.664,E2 -15544.664} C_VEL
LIN {X 0,Y 315.687,Z 340.239,A -85,B 0,C 180,E1 -15545.956,E2 -15545.956} C_VEL
LIN {X 0,Y 321.264,Z 379.585,A -85,B 0,C 180,E1 -15547.241,E2 -15547.241} C_VEL
LIN {X 0,Y 319.959,Z 448.437,A -85,B 0,C 180,E1 -15548.794,E2 -15548.794} C_VEL
LIN {X 0,Y 319.217,Z 461.767,A -85,B 0,C 180,E1 -15549.333,E2 -15549.333} C_VEL
LIN {X 0,Y 318.257,Z 473.981,A -85,B 0,C 180,E1 -15550.069,E2 -15550.069} C_VEL
LIN {X 0,Y 317.166,Z 486.307,A -85,B 0,C 180,E1 -15551.092,E2 -15551.092} C_VEL
LIN {X 0,Y 315.811,Z 497.942,A -85,B 0,C 180,E1 -15552.351,E2 -15552.351} C_VEL
LIN {X 0,Y 314.664,Z 508.646,A -85,B 0,C 180,E1 -15553.822,E2 -15553.822} C_VEL
LIN {X 0,Y 313.588,Z 517.839,A -85,B 0,C 180,E1 -15555.398,E2 -15555.398} C_VEL
LIN {X 0,Y 312.503,Z 526.929,A -85,B 0,C 180,E1 -15557.335,E2 -15557.335} C_VEL
LIN {X 0,Y 311.719,Z 534.243,A -85,B 0,C 180,E1 -15559.281,E2 -15559.281} C_VEL
LIN {X 0,Y 311.258,Z 539.175,A -85,B 0,C 180,E1 -15560.907,E2 -15560.907} C_VEL
LIN {X 0,Y 310.924,Z 543.958,A -85,B 0,C 180,E1 -15562.86,E2 -15562.86} C_VEL
LIN {X 0,Y 310.723,Z 547.603,A -85,B 0,C 180,E1 -15564.81,E2 -15564.81} C_VEL
LIN {X 0,Y 310.724,Z 549.483,A -85,B 0,C 180,E1 -15566.11,E2 -15566.11} C_VEL
LIN {X 0,Y 310.69,Z 550.888,A -85,B 0,C 180,E1 -15567.408,E2 -15567.408} C_VEL
LIN {X 0,Y 310.662,Z 551.884,A -85,B 0,C 180,E1 -15568.705,E2 -15568.705} C_VEL
LIN {X 0,Y 310.693,Z 552.49,A -85,B 0,C 180,E1 -15570.001,E2 -15570.001} C_VEL
LIN {X 0,Y 310.656,Z 552.703,A -85,B 0,C 180,E1 -15571.297,E2 -15571.297} C_VEL
LIN {X 0,Y 310.677,Z 552.486,A -85,B 0,C 180,E1 -15572.594,E2 -15572.594} C_VEL
LIN {X 0,Y 310.699,Z 551.874,A -85,B 0,C 180,E1 -15573.892,E2 -15573.892} C_VEL
LIN {X 0,Y 310.837,Z 549.489,A -85,B 0,C 180,E1 -15576.492,E2 -15576.492} C_VEL
LIN {X 0,Y 311.238,Z 546.575,A -85,B 0,C 180,E1 -15578.441,E2 -15578.441} C_VEL
LIN {X 0,Y 311.856,Z 542.648,A -85,B 0,C 180,E1 -15580.387,E2 -15580.387} C_VEL
LIN {X 0,Y 312.732,Z 537.609,A -85,B 0,C 180,E1 -15582.328,E2 -15582.328} C_VEL
LIN {X 0,Y 314.016,Z 531.3,A -85,B 0,C 180,E1 -15584.253,E2 -15584.253} C_VEL
LIN {X 0,Y 315.627,Z 523.424,A -85,B 0,C 180,E1 -15586.162,E2 -15586.162} C_VEL
LIN {X 0,Y 317.018,Z 515.475,A -85,B 0,C 180,E1 -15587.741,E2 -15587.741} C_VEL
LIN {X 0,Y 318.822,Z 505.704,A -85,B 0,C 180,E1 -15589.309,E2 -15589.309} C_VEL
LIN {X 0,Y 320.71,Z 494.885,A -85,B 0,C 180,E1 -15590.694,E2 -15590.694} C_VEL
LIN {X 0,Y 322.332,Z 484.318,A -85,B 0,C 180,E1 -15591.757,E2 -15591.757} C_VEL
LIN {X 0,Y 323.751,Z 472.76,A -85,B 0,C 180,E1 -15592.664,E2 -15592.664} C_VEL
LIN {X 0,Y 325.137,Z 459.672,A -85,B 0,C 180,E1 -15593.403,E2 -15593.403} C_VEL
LIN {X 0,Y 325.968,Z 446.624,A -85,B 0,C 180,E1 -15593.888,E2 -15593.888} C_VEL
LIN {X 0,Y 327.625,Z 381.25,A -85,B 0,C 180,E1 -15595.36,E2 -15595.36} C_VEL
LIN {X 0,Y 324.738,Z 364.814,A -85,B 0,C 180,E1 -15596.054,E2 -15596.054} C_VEL
LIN {X 0,Y 320.96,Z 347.245,A -85,B 0,C 180,E1 -15596.888,E2 -15596.888} C_VEL
LIN {X 0,Y 317.846,Z 339.531,A -85,B 0,C 180,E1 -15597.45,E2 -15597.45} C_VEL
LIN {X 0,Y 316.008,Z 330.726,A -85,B 0,C 180,E1 -15600.222,E2 -15600.222} C_VEL
LIN {X 0,Y 313.809,Z 321.653,A -85,B 0,C 180,E1 -15603.245,E2 -15603.245} C_VEL
LIN {X 0,Y 312.532,Z 316.56,A -85,B 0,C 180,E1 -15605.089,E2 -15605.089} C_VEL
LIN {X 0,Y 312.497,Z 316.559,A -85,B 0,C 180,E1 -15609.03,E2 -15609.03} C_VEL
LIN {X 0,Y 312.491,Z 316.562,A -85,B 0,C 180,E1 -15612.432,E2 -15612.432} C_VEL
LIN {X 0,Y 312.46,Z 316.561,A -85,B 0,C 180,E1 -15616.035,E2 -15616.035} C_VEL
LIN {X 0,Y 312.505,Z 316.556,A -85,B 0,C 180,E1 -15619.875,E2 -15619.875} C_VEL
LIN {X 0,Y 312.536,Z 316.552,A -85,B 0,C 180,E1 -15624.051,E2 -15624.051} C_VEL
LIN {X 0,Y 312.503,Z 316.552,A -85,B 0,C 180,E1 -15627.334,E2 -15627.334} C_VEL
LIN {X 0,Y 312.526,Z 316.549,A -85,B 0,C 180,E1 -15631.286,E2 -15631.286} C_VEL
LIN {X 0,Y 312.556,Z 316.548,A -85,B 0,C 180,E1 -15634.708,E2 -15634.708} C_VEL
LIN {X 0,Y 312.565,Z 316.55,A -85,B 0,C 180,E1 -15637.527,E2 -15637.527} C_VEL
LIN {X 0,Y 312.569,Z 316.548,A -85,B 0,C 180,E1 -15641.652,E2 -15641.652} C_VEL
LIN {X 0,Y 312.688,Z 316.533,A -85,B 0,C 180,E1 -15645.686,E2 -15645.686} C_VEL
LIN {X 0,Y 312.699,Z 316.533,A -85,B 0,C 180,E1 -15649.642,E2 -15649.642} C_VEL
LIN {X 0,Y 312.893,Z 316.504,A -85,B 0,C 180,E1 -15653.552,E2 -15653.552} C_VEL
LIN {X 0,Y 312.984,Z 316.492,A -85,B 0,C 180,E1 -15658.714,E2 -15658.714} C_VEL
LIN {X 0,Y 312.985,Z 316.488,A -85,B 0,C 180,E1 -15661.287,E2 -15661.287} C_VEL
LIN {X 0,Y 312.703,Z 316.523,A -85,B 0,C 180,E1 -15665.158,E2 -15665.158} C_VEL
LIN {X 0,Y 312.82,Z 316.516,A -85,B 0,C 180,E1 -15667.747,E2 -15667.747} C_VEL
LIN {X 0,Y 312.666,Z 316.536,A -85,B 0,C 180,E1 -15671.672,E2 -15671.672} C_VEL
LIN {X 0,Y 312.67,Z 316.537,A -85,B 0,C 180,E1 -15674.865,E2 -15674.865} C_VEL
LIN {X 0,Y 312.591,Z 316.547,A -85,B 0,C 180,E1 -15679.214,E2 -15679.214} C_VEL
LIN {X 0,Y 312.528,Z 316.551,A -85,B 0,C 180,E1 -15682.78,E2 -15682.78} C_VEL
LIN {X 0,Y 312.541,Z 316.548,A -85,B 0,C 180,E1 -15685.911,E2 -15685.911} C_VEL
LIN {X 0,Y 312.507,Z 316.557,A -85,B 0,C 180,E1 -15689.654,E2 -15689.654} C_VEL
LIN {X 0,Y 312.523,Z 316.553,A -85,B 0,C 180,E1 -15693.689,E2 -15693.689} C_VEL
LIN {X 0,Y 312.529,Z 316.552,A -85,B 0,C 180,E1 -15697.385,E2 -15697.385} C_VEL
LIN {X 0,Y 312.493,Z 316.56,A -85,B 0,C 180,E1 -15700.709,E2 -15700.709} C_VEL
LIN {X 0,Y 312.455,Z 316.563,A -85,B 0,C 180,E1 -15704.21,E2 -15704.21} C_VEL
LIN {X 0,Y 312.459,Z 316.566,A -85,B 0,C 180,E1 -15707.925,E2 -15707.925} C_VEL
LIN {X 0,Y 312.499,Z 316.757,A -85,B 0,C 180,E1 -15708.487,E2 -15708.487} C_VEL
LIN {X 0,Y 314.575,Z 324.657,A -85,B 0,C 180,E1 -15711.251,E2 -15711.251} C_VEL
LIN {X 0,Y 323.266,Z 343.121,A -85,B 0,C 180,E1 -15712.676,E2 -15712.676} C_VEL
LIN {X 0,Y 327.111,Z 352.29,A -85,B 0,C 180,E1 -15713.299,E2 -15713.299} C_VEL
LIN {X 0,Y 328.344,Z 358.83,A -85,B 0,C 180,E1 -15713.584,E2 -15713.584} C_VEL
LIN {X 0,Y 326.195,Z 432.605,A -85,B 0,C 180,E1 -15715.24,E2 -15715.24} C_VEL
LIN {X 0,Y 325.384,Z 444.807,A -85,B 0,C 180,E1 -15715.731,E2 -15715.731} C_VEL
LIN {X 0,Y 324.123,Z 458.07,A -85,B 0,C 180,E1 -15716.525,E2 -15716.525} C_VEL
LIN {X 0,Y 322.921,Z 468.773,A -85,B 0,C 180,E1 -15717.407,E2 -15717.407} C_VEL
LIN {X 0,Y 321.319,Z 480.55,A -85,B 0,C 180,E1 -15718.666,E2 -15718.666} C_VEL
LIN {X 0,Y 319.439,Z 491.534,A -85,B 0,C 180,E1 -15720.146,E2 -15720.146} C_VEL
LIN {X 0,Y 317.773,Z 500.234,A -85,B 0,C 180,E1 -15721.607,E2 -15721.607} C_VEL
LIN {X 0,Y 316.2,Z 508.427,A -85,B 0,C 180,E1 -15723.31,E2 -15723.31} C_VEL
LIN {X 0,Y 314.613,Z 515.907,A -85,B 0,C 180,E1 -15725.237,E2 -15725.237} C_VEL
LIN {X 0,Y 313.209,Z 522.977,A -85,B 0,C 180,E1 -15727.575,E2 -15727.575} C_VEL
LIN {X 0,Y 312.212,Z 527.579,A -85,B 0,C 180,E1 -15729.579,E2 -15729.579} C_VEL
LIN {X 0,Y 311.563,Z 531.038,A -85,B 0,C 180,E1 -15731.59,E2 -15731.59} C_VEL
LIN {X 0,Y 311.159,Z 532.737,A -85,B 0,C 180,E1 -15732.924,E2 -15732.924} C_VEL
LIN {X 0,Y 310.897,Z 534.018,A -85,B 0,C 180,E1 -15734.26,E2 -15734.26} C_VEL
LIN {X 0,Y 310.722,Z 535.232,A -85,B 0,C 180,E1 -15736.556,E2 -15736.556} C_VEL
LIN {X 0,Y 310.589,Z 535.312,A -85,B 0,C 180,E1 -15738.249,E2 -15738.249} C_VEL
LIN {X 0,Y 310.497,Z 534.938,A -85,B 0,C 180,E1 -15739.567,E2 -15739.567} C_VEL
LIN {X 0,Y 310.55,Z 534.158,A -85,B 0,C 180,E1 -15740.884,E2 -15740.884} C_VEL
LIN {X 0,Y 310.642,Z 532.932,A -85,B 0,C 180,E1 -15742.197,E2 -15742.197} C_VEL
LIN {X 0,Y 310.877,Z 530.418,A -85,B 0,C 180,E1 -15744.109,E2 -15744.109} C_VEL
LIN {X 0,Y 311.164,Z 526.731,A -85,B 0,C 180,E1 -15746.114,E2 -15746.114} C_VEL
LIN {X 0,Y 311.606,Z 522.022,A -85,B 0,C 180,E1 -15748.06,E2 -15748.06} C_VEL
